(* CoDeSys 2.3.9.41 project: 5AxisMachine.pro *)
(* Libraries: TcUtilities.lib 10.1.13 20:12:12, TcBase.lib 14.5.09 12:14:08, TcSystem.lib 16.1.14 19:38:48, TcBaseMath.lib 27.7.04 12:07:56, TcMath.lib 23.9.04 15:15:30, TcMC2.lib 14.7.14 11:34:46, STANDARD.LIB 5.6.98 12:03:02, TcSUPS.lib 22.3.10 13:59:22, SysLibVisu.lib 7.7.04 18:17:22, SysLibTargetVisu.lib 16.6.08 16:24:26 *)

(* Task configuration *)
TASK Standard (PRIORITY := 0, INTERVAL := T#10ms);
	MAIN
END_TASK
TASK VISU_TASK (PRIORITY := 3, INTERVAL := T#200ms);
	MAINTARGETVISU_PAINT_CODE
END_TASK
TASK VISU_INPUT_TASK (PRIORITY := 2, INTERVAL := T#50ms);
	MAINTARGETVISU_INPUT_CODE
END_TASK

(* Global variable list: Global1_Persistent_Variables *)
VAR_GLOBAL PERSISTENT
	MachineRecipes				: ARRAY[1..NUMBER_OF_RECIPES] OF Recipe;
	nCurrentRecipe				: BYTE := 1; (* Current Machine Recipe *)
	nPartsCounter				: DWORD;


	VisuDoExecuteUserlevelInit 	: BOOL := TRUE;
	CurrentUserLevel 			: INT := 0;
	CurrentPasswords 			: ARRAY[0..7] OF STRING[20] := '','1','2','3','superuser4','8600','arl6','arl7'; (* Assigns Password Defaults *)
END_VAR

(* Global variable list: Global_Constant *)
VAR_GLOBAL CONSTANT
	NUMBER_OF_AXIS		: BYTE := 5;
	NUMBER_OF_MOVES 	: BYTE := 9;
	NUMBER_OF_RECIPES 	: BYTE := 25;
	CUTTER				: BYTE := 1;
	SIZER				: BYTE := 2;

	LEFT_HAND_SPINDLE	: BYTE := 1;
	RIGHT_HAND_SPINDLE	: BYTE := 2;
	CUTTER_AXIS			: BYTE := 3;
	CUTTER_SLIDE		: BYTE := 4;
	ENGAGE_AXIS			: BYTE := 5;

	SIZER_AXIS			: BYTE := 1;
	ARBOR_AXIS			: BYTE := 2;

	MAX_CYCLE_TIME		: WORD := 120;


	DEAFULT_AXIS_SPEED	: LREAL := 500;

	VERSION_NUMBER		: STRING :='V1.0.0 9_19_14';



END_VAR

(* Global variable list: Global_Variables *)
VAR_GLOBAL

(* IO Defined Here *)
	nRecipeNumber							   : BYTE; (* Holds Recipe Number for Editor *)

	Faults									   : Faults_STRUCT;
	Warnings								   : Warnings_STRUCT;

	nMachineType							   : BYTE := SIZER; (* Defines Machine Type 1 = Cutter, 2 = Sizer *)
	bAutomaticMode							   : BOOL;
END_VAR

(* Global variable list: Global_Variables_IO *)
VAR_GLOBAL
	(************ INPUTS ***********************)
	ibPowerOn						AT %I*		: BOOL;			(* True when power is on						*)
	ibLightScreenClear				AT %I*		: BOOL;			(* True when light screen is clear				*)
	ibCycleStartPB					AT %I*		: BOOL;			(* when true start machine cycle				*)
	ibLeftHandSpindleDriveOn		AT %I*		: BOOL;			(* When true left hand spindle is on			*)
	ibLeftHandSpindleDriveOK		AT %I*		: BOOL;			(* When true left hand spindle drive is faulted	*)
	ibRightHandSpindleDriveOn		AT %I*		: BOOL;			(* When true right hand spindle is on			*)
	ibRightHandSpindleDriveOK		AT %I*		: BOOL;			(* When true right hand spindle drive is faulted*)
	ibPartClampAdvanced				AT %I*		: BOOL;			(* When true the part clamp is clamped  		*)
	ibPartClampReturned				AT %I*		: BOOL;			(* When true the part clamp is returned 		*)
	ibPartClampLocked				AT %I*		: BOOL;			(* When true part clamp is in locked position	*)
	ibHydraulicsOverload			AT %I*		: BOOL;			(* Hydraulics overloaded when false				*)
	ibHydraulicsOverTemp			AT %I*		: BOOL;			(* Hydraulics over temp							*)
	ibHydraulicsLowLevel			AT %I*		: BOOL;			(* Hydraulics low level							*)

	(*************OUTPUTS***********************)

	qbLeftHandSpindleOn				AT %Q*		: BOOL;			(* Enable left hand spindle						*)
	qbRightHandSpindleOn			AT %Q*		: BOOL;			(* Enable right hand spindle					*)
	qbClosePartClampSolA			AT %Q*		: BOOL;			(* When true part clamp solenoid A closes clamp	*)
	qbOpenPartClampSolB				AT %Q*		: BOOL;			(* When trie part clamp solendoid B opens clamp *)
	qbSpareOutput					AT %Q*		: BOOL;
	qbOKToEnterGreenLamp			AT %Q*		: BOOL;
	qbMachineInCycleFaultRedLamp	AT %Q*		: BOOL;


END_VAR

(* Global variable list: TwinCAT_Configuration *)
(* Generated automatically by TwinCAT - (read only) *)
VAR_CONFIG
	MAIN.Axis_REF[1].PlcToNc AT %QB1 : PLCTONC_AXIS_REF;
	MAIN.Axis_REF[1].NcToPlc AT %IB6 : NCTOPLC_AXIS_REF;
	MAIN.Axis_REF[2].PlcToNc AT %QB129 : PLCTONC_AXIS_REF;
	MAIN.Axis_REF[2].NcToPlc AT %IB134 : NCTOPLC_AXIS_REF;
	MAIN.Axis_REF[3].PlcToNc AT %QB257 : PLCTONC_AXIS_REF;
	MAIN.Axis_REF[3].NcToPlc AT %IB262 : NCTOPLC_AXIS_REF;
	MAIN.Axis_REF[4].PlcToNc AT %QB385 : PLCTONC_AXIS_REF;
	MAIN.Axis_REF[4].NcToPlc AT %IB390 : NCTOPLC_AXIS_REF;
	MAIN.Axis_REF[5].PlcToNc AT %QB513 : PLCTONC_AXIS_REF;
	MAIN.Axis_REF[5].NcToPlc AT %IB518 : NCTOPLC_AXIS_REF;
	.ibPowerOn AT %IX648.0 : BOOL;	(*  ~ {LinkedWith:TIID^Device 1 (EtherCAT)^Term 1 (EK1200)^Term 2 (EL1809)^Channel 1^Power On} *)
	.ibLightScreenClear AT %IX648.1 : BOOL;	(*  ~ {LinkedWith:TIID^Device 1 (EtherCAT)^Term 1 (EK1200)^Term 2 (EL1809)^Channel 2^Light Curtain Clear} *)
	.ibCycleStartPB AT %IX648.2 : BOOL;	(*  ~ {LinkedWith:TIID^Device 1 (EtherCAT)^Term 1 (EK1200)^Term 2 (EL1809)^Channel 3^Cycle Start} *)
	.ibLeftHandSpindleDriveOn AT %IX648.3 : BOOL;
	.ibLeftHandSpindleDriveOK AT %IX648.4 : BOOL;
	.ibRightHandSpindleDriveOn AT %IX648.5 : BOOL;
	.ibRightHandSpindleDriveOK AT %IX648.6 : BOOL;
	.ibPartClampAdvanced AT %IX648.7 : BOOL;	(*  ~ {LinkedWith:TIID^Device 1 (EtherCAT)^Term 1 (EK1200)^Term 2 (EL1809)^Channel 4^Part Clamp Closed} *)
	.ibPartClampReturned AT %IX649.0 : BOOL;	(*  ~ {LinkedWith:TIID^Device 1 (EtherCAT)^Term 1 (EK1200)^Term 2 (EL1809)^Channel 5^Part Clamp Open} *)
	.ibPartClampLocked AT %IX649.1 : BOOL;
	.ibHydraulicsOverload AT %IX649.2 : BOOL;
	.ibHydraulicsOverTemp AT %IX652.0 : BOOL;
	.ibHydraulicsLowLevel AT %IX652.1 : BOOL;
	.qbLeftHandSpindleOn AT %QX644.0 : BOOL;
	.qbRightHandSpindleOn AT %QX644.1 : BOOL;
	.qbClosePartClampSolA AT %QX644.2 : BOOL;
	.qbOpenPartClampSolB AT %QX644.3 : BOOL;
	.qbSpareOutput AT %QX644.4 : BOOL;
	.qbOKToEnterGreenLamp AT %QX644.5 : BOOL;	(*  ~ {LinkedWith:TIID^Device 1 (EtherCAT)^Term 1 (EK1200)^Term 3 (EL2828)^Channel 7^Green Lamp (OK To Enter)} *)
	.qbMachineInCycleFaultRedLamp AT %QX644.6 : BOOL;	(*  ~ {LinkedWith:TIID^Device 1 (EtherCAT)^Term 1 (EK1200)^Term 3 (EL2828)^Channel 8^Red Lamp (Faulted)} *)
END_VAR

(* Data type *)
TYPE AXISSEQUENCE :
(
	AXIS_INIT,
	AXIS_RESET,
	AXIS_FAULTED,
	AXIS_READY,
	AXIS_POWER_ON,
	AXIS_STOP,
	AXIS_HOMING,
	AXIS_HOMED,
	AXIS_RUNNING
);

END_TYPE

(* Data type *)
TYPE FAULTS_STRUCT :
STRUCT
	bOperator_Stop					: BOOL; (* True when operate stops the machine							*)
	bLeftHandSpindleVFDError		: BOOL; (* True when left hand spindle VFD is at Fault					*)
	bRightHandSpindleVFDError		: BOOL;
	bProgramError					: BOOL;
	bLeftSpindleServoError			: BOOL;
	bRightSpindlervoError			: BOOL;
	bCutterServorError				: BOOL;
	bCutterSlideServoError			: BOOL;
	bEngageServoError				: BOOL;
	bCycleTimeExceeded				: BOOL; (* True when the cycle time took too long to complete			*)
END_STRUCT
END_TYPE

(* Data type *)
TYPE MACHINE_SEQUENCE :
(
	MACHINE_INIT,
	MACHINE_RESET,
	MACHINE_FAULTED,
	MACHINE_READY,
	ENABLE_SERVOS,
	MOVE_TO_END_CUT,
	MOVE_TO_START_SIZER,
	POSITION_SIZER_SERVOS,
	MOVE_TO_CRUSHED_POSITION,
	MOVE_SIZER_TO_RELIEVED_POSITION,
	MOVE_SIZER_TO_UNLOAD,
	RETURN_SIZER,
	MOVE_TO_FIRST_CUT,
	COUPLE_DRIVES,
	DECOUPLE_DRIVES,
	OPERATE_FIRST_CUT,
	MOVE_TO_NEXT_CUT,
	ADVANCE_ENGAGE,
	RETURN_ENGAGE,
	OPERATE_CUT,
	RETRACT_FROM_CUT,
	RETURN_MACHINE
);

END_TYPE

(* Data type *)
TYPE RECIPE :
STRUCT

	bPartClampEnable		: BOOL;											(* When true part clamp is enabled						*)
	arrAxis1MoveTable		: ARRAY[1..NUMBER_OF_MOVES] OF LREAL;			(* Left Spindle Axis move table							*)
	arrAxis2MoveTable		: ARRAY[1..NUMBER_OF_MOVES] OF LREAL;			(* Right spindle move table								*)
	arrAxis3MoveTable		: ARRAY[1..2] OF LREAL;							(* Cutter move table									*)
	arrAxis4MoveTable		: ARRAY[1..NUMBER_OF_MOVES] OF LREAL;			(* Cutter slide move table								*)
	arrAxis5MoveTable		: ARRAY[1..2] OF LREAL;							(* Engage move table									*)
	Axis1HomePosition		: LREAL;										(* Axis 1 Home Position									*)
	nNumberOfCuts			: BYTE;											(* Number of cuts to be made							*)
	timeCutterTimer			: TIME;											(* Cutter Timer Time									*)
	rAxis1Speed				: LREAL;										(* Speed of Axis #1										*)
	rAxis2Speed				: LREAL;										(* Speed of Axis #2										*)
	rAxis3Speed				: LREAL;										(* Speed of Axis #3										*)
	rAxis4Speed				: LREAL;										(* Speed of Axis #4										*)
	rAxis5Speed				: LREAL;										(* Speed of Axis #5										*)
	nNumberOfCycles			: BYTE; 										(* Number of cycles of the sizer						*)
	sRecipeName				: STRING;										(* Part Type Description								*)
END_STRUCT
END_TYPE

(* Data type *)
TYPE WARNINGS_STRUCT :
STRUCT
	bHopperLow						: BOOL;
	bConveyorFull					: BOOL;
END_STRUCT
END_TYPE

(* POU MAIN, LD *)
(********************************************************************************************************
NAME...........	:	Main Program
DATE...........	:	08.6.2014
AUTHOR.........	:	ARL

DESCRIPTION....	:	Handling of main routine for the Machine.

HISTORY:	
08.6.2014	v1.0.0	GPK	Start coding
*********************************************************************************************************)
PROGRAM MAIN
VAR_INPUT
	nTargetPosition 			: ARRAY[1..NUMBER_OF_AXIS] OF LREAL;
	nMoveVelocity   			: ARRAY[1..NUMBER_OF_AXIS] OF LREAL;
	bClosePartClamp				: BOOL;
	bMoveAbsolute				: ARRAY[1..NUMBER_OF_AXIS] OF BOOL;
	bAxisEnable 				: ARRAY[1..NUMBER_OF_AXIS] OF BOOL;


	bLeftHandSpindleRun			: BOOL;
	bRightHandSpindleRun		: BOOL;

	bCoupleAxis					: BOOL;
	bDeCoupleAxis				: BOOL;
	bAxis2Coupled				: BOOL;
	bAxis4Coupled				: BOOL;
	bInCycle					: BOOL;

	bJogAxisForward				: ARRAY[1..NUMBER_OF_AXIS] OF BOOL;
	bJogAxisReverse				: ARRAY[1..NUMBER_OF_AXIS] OF BOOL;
	bFaultPresent				: BOOL;
END_VAR
VAR
	Axis						: ARRAY[1..NUMBER_OF_AXIS] OF FB_Motion;

	Axis_REF					: ARRAY[1..NUMBER_OF_AXIS] OF AXIS_REF;

	bAxisHasError				: ARRAY[1..NUMBER_OF_AXIS] OF BOOL;
	bMoveRelative				: ARRAY[1..NUMBER_OF_AXIS] OF BOOL;
	bMoveComplete				: ARRAY[1..NUMBER_OF_AXIS] OF BOOL;
	bPowerOnActive				: ARRAY[1..NUMBER_OF_AXIS] OF BOOL;


	sSequenceText				: ARRAY[1..NUMBER_OF_AXIS] OF STRING;
	loop						: BYTE; (* Used to loop through all axis *)
	bResetLoop					: BOOL;


	bStartMachine				: BOOL;
	bStopMachine				: BOOL;
	bReset						: BOOL;
	bMachineRunning				: BOOL;





	ToggleLamp					: FB_Toggle; 			(* FB to toggle variable or output off/on   *)
	LeftHandSpindleMotor		: FB_Motor_Ctrl; 		(* FB for simple motor control 				*)
	RightHandSpindleMotor		: FB_Motor_Ctrl; 		(* FB for simple motor control 				*)
	PartClamp					: FB_CylinderControl;	(* FB To Operate Part Clamp					*)

	ctCycleCounter				: CTU;
	wCounterPreset				: WORD; (* Some Comment *)


	bResetCounter				: BOOL;		(*Reset Counter*)
	bTriggerCounter				: BOOL;
	CounterDone					: BOOL;
	bStartButtonIndicator		: BOOL;
	bResetTimeCounter			: BOOL;


	CoupleAxis2					: FB_CoupleAxis;
	CoupleAxis4					: FB_CoupleAxis;

	tmrCycleTimer				: TON;

	cntSecondsCounter			: CTU;
	re_InCycle					: R_TRIG;
	nCycleTime					: WORD;

END_VAR
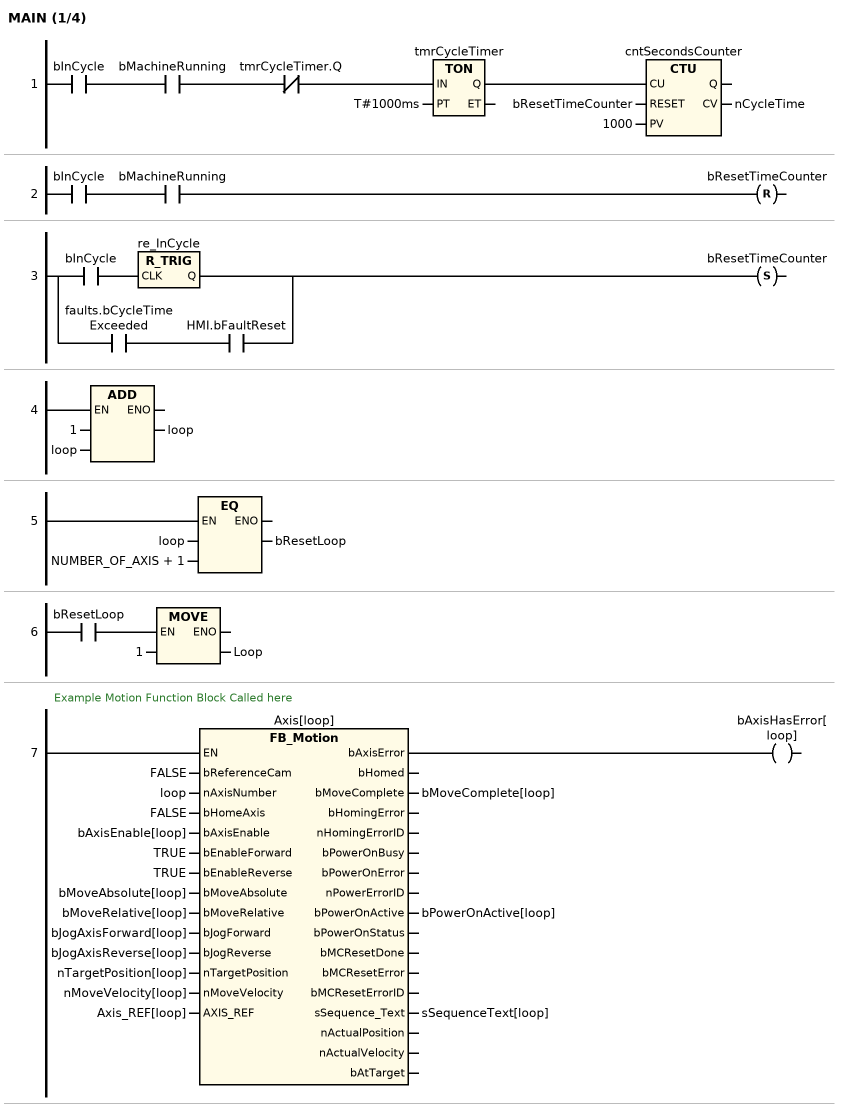
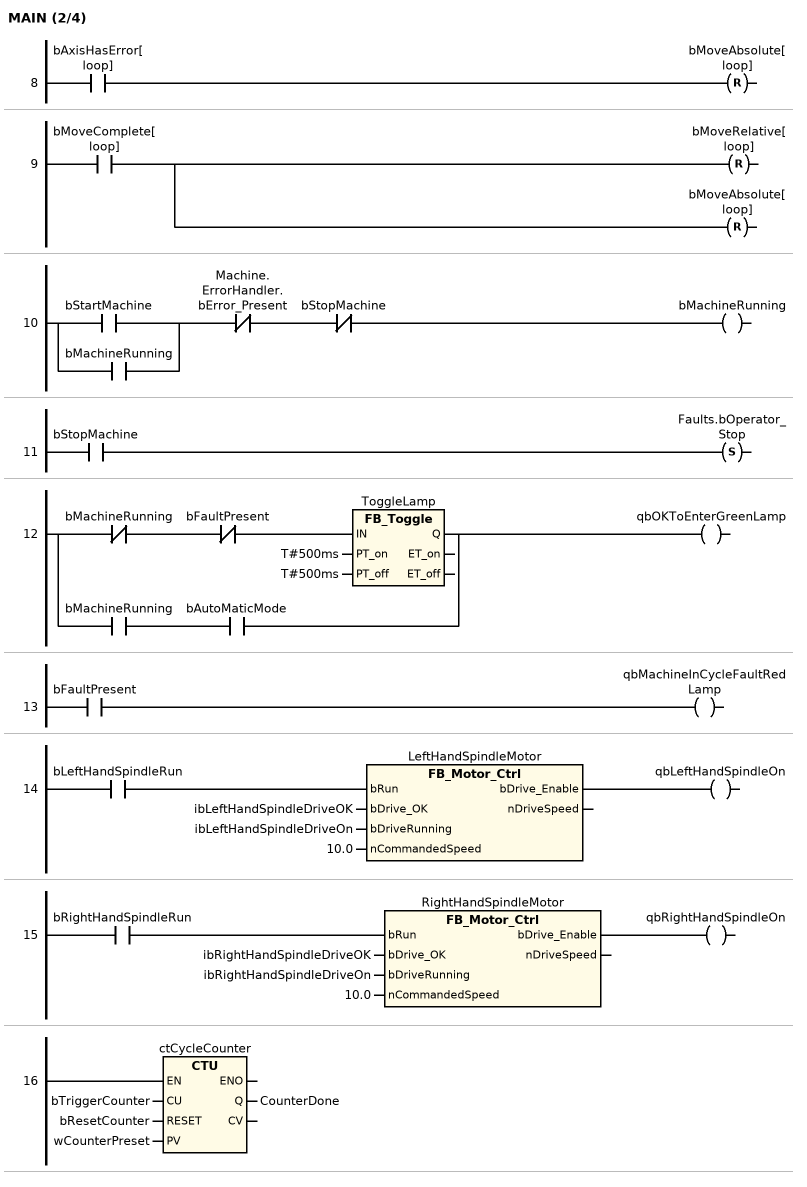
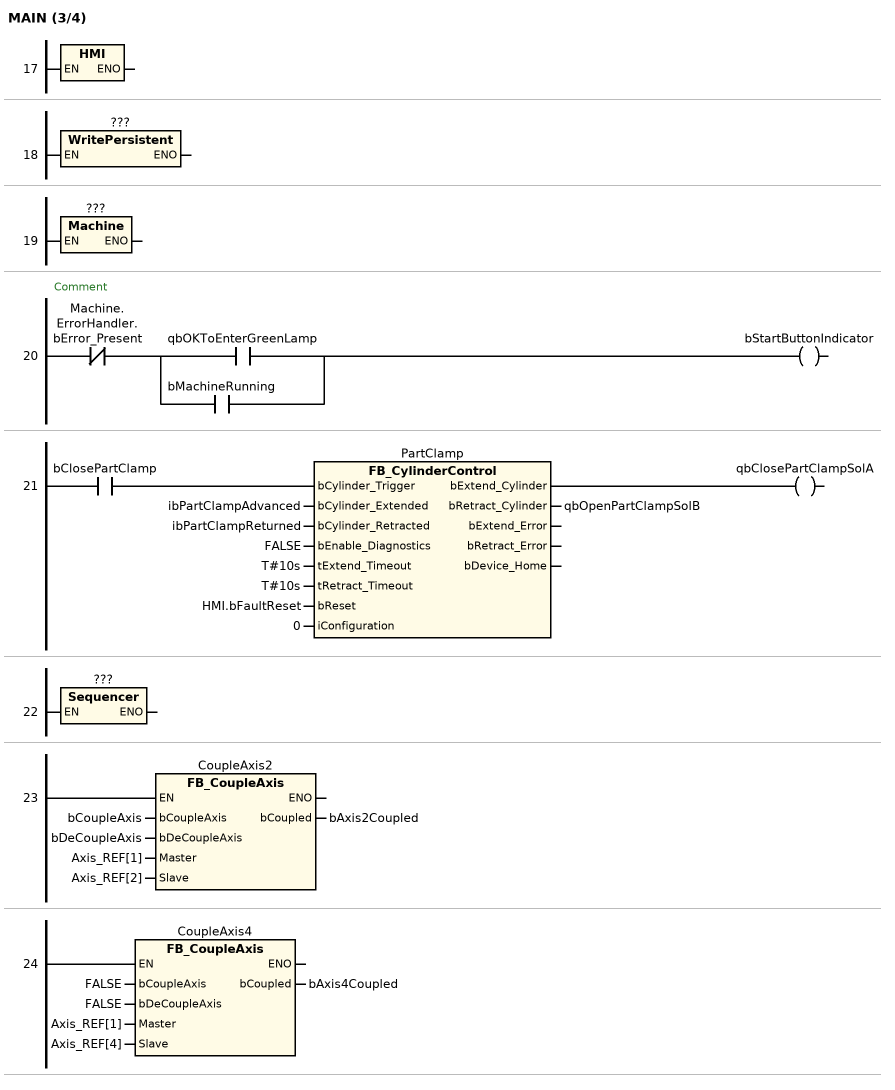
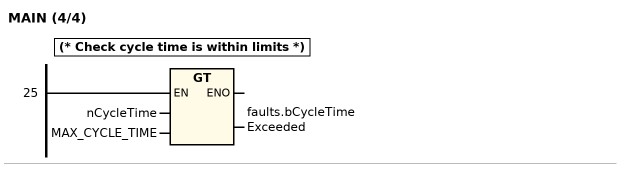
_LD_ (* Ladder Diagram *)
NETWORK 1
	[bInCycle] - [bMachineRunning] - [/tmrCycleTimer.Q] - tmrCycleTimer:TON(IN: *, PT: T#1000ms) - cntSecondsCounter:CTU(CU: *, RESET: bResetTimeCounter, PV: 1000, CV => nCycleTime)
NETWORK 2
	[bInCycle] - [bMachineRunning] --- (R bResetTimeCounter)
NETWORK 3
	{ [bInCycle] - re_InCycle:R_TRIG(CLK: *) | [faults.bCycleTimeExceeded] - [HMI.bFaultReset] } --- (S bResetTimeCounter)
NETWORK 4
	*
		EN --- ADD(1, loop) => loop
NETWORK 5
	*
		EN --- EQ(loop, NUMBER_OF_AXIS + 1) => bResetLoop
NETWORK 6
	[bResetLoop]
		EN --- MOVE(1) => Loop
NETWORK 7 (* Example Motion Function Block Called here *)
	Axis[loop]:FB_Motion(EN: *, bReferenceCam: FALSE, nAxisNumber: loop, bHomeAxis: FALSE, bAxisEnable: bAxisEnable[loop], bEnableForward: TRUE, bEnableReverse: TRUE, bMoveAbsolute: bMoveAbsolute[loop], bMoveRelative: bMoveRelative[loop], bJogForward: bJogAxisForward[loop], bJogReverse: bJogAxisReverse[loop], nTargetPosition: nTargetPosition[loop], nMoveVelocity: nMoveVelocity[loop], AXIS_REF: Axis_REF[loop], bMoveComplete => bMoveComplete[loop], bPowerOnActive => bPowerOnActive[loop], sSequence_Text => sSequenceText[loop]) --- (bAxisHasError[loop])
NETWORK 8
	[bAxisHasError[loop]] --- (R bMoveAbsolute[loop])
NETWORK 9
	[bMoveComplete[loop]] --- (R bMoveRelative[loop]) (R bMoveAbsolute[loop])
NETWORK 10
	{ [bStartMachine] | [bMachineRunning] } - [/Machine.ErrorHandler.bError_Present] - [/bStopMachine] --- (bMachineRunning)
NETWORK 11
	[bStopMachine] --- (S Faults.bOperator_Stop)
NETWORK 12
	{ [/bMachineRunning] - [/bFaultPresent] - ToggleLamp:FB_Toggle(IN: *, PT_on: T#500ms, PT_off: T#500ms) | [bMachineRunning] - [bAutoMaticMode] } --- (qbOKToEnterGreenLamp)
NETWORK 13
	[bFaultPresent] --- (qbMachineInCycleFaultRedLamp)
NETWORK 14
	[bLeftHandSpindleRun] - LeftHandSpindleMotor:FB_Motor_Ctrl(bRun: *, bDrive_OK: ibLeftHandSpindleDriveOK, bDriveRunning: ibLeftHandSpindleDriveOn, nCommandedSpeed: 10.0) --- (qbLeftHandSpindleOn)
NETWORK 15
	[bRightHandSpindleRun] - RightHandSpindleMotor:FB_Motor_Ctrl(bRun: *, bDrive_OK: ibRightHandSpindleDriveOK, bDriveRunning: ibRightHandSpindleDriveOn, nCommandedSpeed: 10.0) --- (qbRightHandSpindleOn)
NETWORK 16
	*
		EN --- ctCycleCounter:CTU(CU: bTriggerCounter, RESET: bResetCounter, PV: wCounterPreset) => CounterDone
NETWORK 17
	*
		EN --- HMI()
NETWORK 18
	*
		EN --- ???:WritePersistent()
NETWORK 19
	*
		EN --- ???:Machine()
NETWORK 20 (* Comment *)
	[/Machine.ErrorHandler.bError_Present] - { [qbOKToEnterGreenLamp] | [bMachineRunning] } --- (bStartButtonIndicator)
NETWORK 21
	[bClosePartClamp] - PartClamp:FB_CylinderControl(bCylinder_Trigger: *, bCylinder_Extended: ibPartClampAdvanced, bCylinder_Retracted: ibPartClampReturned, bEnable_Diagnostics: FALSE, tExtend_Timeout: T#10s, tRetract_Timeout: T#10s, bReset: HMI.bFaultReset, iConfiguration: 0, bRetract_Cylinder => qbOpenPartClampSolB) --- (qbClosePartClampSolA)
NETWORK 22
	*
		EN --- ???:Sequencer()
NETWORK 23
	*
		EN --- CoupleAxis2:FB_CoupleAxis(bCoupleAxis: bCoupleAxis, bDeCoupleAxis: bDeCoupleAxis, Master: Axis_REF[1], Slave: Axis_REF[2]) => bAxis2Coupled
NETWORK 24
	*
		EN --- CoupleAxis4:FB_CoupleAxis(bCoupleAxis: FALSE, bDeCoupleAxis: FALSE, Master: Axis_REF[1], Slave: Axis_REF[4]) => bAxis4Coupled
NETWORK 25 (* Check cycle time is within limits *):
	*
		EN --- GT(nCycleTime, MAX_CYCLE_TIME) => faults.bCycleTimeExceeded
_END_LD_
(* the same logic as Structured Text *)
(* Network 1 *)
tmrCycleTimer(IN := bInCycle AND bMachineRunning AND NOT tmrCycleTimer.Q, PT := T#1000ms);
cntSecondsCounter(CU := tmrCycleTimer.Q, RESET := bResetTimeCounter, PV := 1000);
nCycleTime := cntSecondsCounter.CV;
(* Network 2 *)
IF bInCycle AND bMachineRunning THEN bResetTimeCounter := FALSE; END_IF;
(* Network 3 *)
re_InCycle(CLK := bInCycle);
IF re_InCycle.Q OR faults.bCycleTimeExceeded AND HMI.bFaultReset THEN bResetTimeCounter := TRUE; END_IF;
(* Network 4 *)
loop := 1 + loop;
(* Network 5 *)
bResetLoop := loop = (NUMBER_OF_AXIS + 1);
(* Network 6 *)
IF bResetLoop THEN
	Loop := 1;
END_IF;
(* Network 7 *)
Axis[loop](EN := TRUE, bReferenceCam := FALSE, nAxisNumber := loop, bHomeAxis := FALSE, bAxisEnable := bAxisEnable[loop], bEnableForward := TRUE, bEnableReverse := TRUE, bMoveAbsolute := bMoveAbsolute[loop], bMoveRelative := bMoveRelative[loop], bJogForward := bJogAxisForward[loop], bJogReverse := bJogAxisReverse[loop], nTargetPosition := nTargetPosition[loop], nMoveVelocity := nMoveVelocity[loop], AXIS_REF := Axis_REF[loop]);
bMoveComplete[loop] := Axis[loop].bMoveComplete;
bPowerOnActive[loop] := Axis[loop].bPowerOnActive;
sSequenceText[loop] := Axis[loop].sSequence_Text;
bAxisHasError[loop] := Axis[loop].bAxisError;
(* Network 8 *)
IF bAxisHasError[loop] THEN bMoveAbsolute[loop] := FALSE; END_IF;
(* Network 9 *)
IF bMoveComplete[loop] THEN bMoveRelative[loop] := FALSE; bMoveAbsolute[loop] := FALSE; END_IF;
(* Network 10 *)
bMachineRunning := (bStartMachine OR bMachineRunning) AND NOT Machine.ErrorHandler.bError_Present AND NOT bStopMachine;
(* Network 11 *)
IF bStopMachine THEN Faults.bOperator_Stop := TRUE; END_IF;
(* Network 12 *)
ToggleLamp(IN := NOT bMachineRunning AND NOT bFaultPresent, PT_on := T#500ms, PT_off := T#500ms);
qbOKToEnterGreenLamp := ToggleLamp.Q OR bMachineRunning AND bAutoMaticMode;
(* Network 13 *)
qbMachineInCycleFaultRedLamp := bFaultPresent;
(* Network 14 *)
LeftHandSpindleMotor(bRun := bLeftHandSpindleRun, bDrive_OK := ibLeftHandSpindleDriveOK, bDriveRunning := ibLeftHandSpindleDriveOn, nCommandedSpeed := 10.0);
qbLeftHandSpindleOn := LeftHandSpindleMotor.bDrive_Enable;
(* Network 15 *)
RightHandSpindleMotor(bRun := bRightHandSpindleRun, bDrive_OK := ibRightHandSpindleDriveOK, bDriveRunning := ibRightHandSpindleDriveOn, nCommandedSpeed := 10.0);
qbRightHandSpindleOn := RightHandSpindleMotor.bDrive_Enable;
(* Network 16 *)
ctCycleCounter(CU := bTriggerCounter, RESET := bResetCounter, PV := wCounterPreset);
CounterDone := ctCycleCounter.Q;
(* Network 17 *)
HMI();
(* Network 18: see the listing above *)
(* Network 19: see the listing above *)
(* Network 20 *)
bStartButtonIndicator := NOT Machine.ErrorHandler.bError_Present AND (qbOKToEnterGreenLamp OR bMachineRunning);
(* Network 21 *)
PartClamp(bCylinder_Trigger := bClosePartClamp, bCylinder_Extended := ibPartClampAdvanced, bCylinder_Retracted := ibPartClampReturned, bEnable_Diagnostics := FALSE, tExtend_Timeout := T#10s, tRetract_Timeout := T#10s, bReset := HMI.bFaultReset, iConfiguration := 0);
qbOpenPartClampSolB := PartClamp.bRetract_Cylinder;
qbClosePartClampSolA := PartClamp.bExtend_Cylinder;
(* Network 22: see the listing above *)
(* Network 23 *)
CoupleAxis2(bCoupleAxis := bCoupleAxis, bDeCoupleAxis := bDeCoupleAxis, Master := Axis_REF[1], Slave := Axis_REF[2]);
bAxis2Coupled := CoupleAxis2.bCoupled;
(* Network 24 *)
CoupleAxis4(bCoupleAxis := FALSE, bDeCoupleAxis := FALSE, Master := Axis_REF[1], Slave := Axis_REF[4]);
bAxis4Coupled := CoupleAxis4.bCoupled;
(* Network 25 *)
faults.bCycleTimeExceeded := nCycleTime > MAX_CYCLE_TIME;
END_PROGRAM

(* POU Motion/FB_Motion, ST *)
(********************************************************************************************************

NAME...........	:	FB_Motion
DATE...........	:	7/23/2014
AUTHOR.........	:	Graeme Peek Beckhoff Automation

DESCRIPTION....	:	Motion Axis Control Function Block
					NOTE: Given as is as an example, if used as part of a working machine then it must be validated and adjusted as required.
					Beckhoff assumes no responsability for the accuracy of this software.

HISTORY:	
5/23/2014	v1.0.0	Graeme	Start coding
*************************************************************************************************************)
FUNCTION_BLOCK FB_Motion
VAR_INPUT
	EN						: BOOL;						(* Block enabled when true							*)
	bReferenceCam			: BOOL; 					(* True when reference cam is on 					*)
	nAxisNumber				: BYTE;						(* Holds Axis Number								*)
	bHomeAxis				: BOOL;						(* When true homing is initiated					*)
	bAxisEnable				: BOOL;						(* When true then enable this axis					*)
	bEnableForward			: BOOL;
	bEnableReverse			: BOOL;
	bMoveAbsolute			: BOOL;
	bMoveRelative			: BOOL;
	bJogForward				: BOOL;						(* When true axis jogs forward						*)
	bJogReverse				: BOOL;						(* When true axis jogs in reverse					*)
	nTargetPosition			: LREAL;
	nMoveVelocity			: LREAL;
END_VAR
VAR_OUTPUT
	bAxisError				: BOOL;
	bHomed					: BOOL;						(* True when axis has homed							*)
	bMoveComplete			: BOOL;						(* True when any move has completed					*)
	bHomingError			: BOOL;						(* True when an error ocurred to the homing FB		*)
	nHomingErrorID			: UDINT;					(* Holds homing FB error code						*)
	bPowerOnBusy			: BOOL;						(* True when power is on 							*)
	bPowerOnError			: BOOL;						(* True if an error occurred turing axis power on	*)
	nPowerErrorID			: UDINT;					(* Holds error code for power on command			*)
	bPowerOnActive			: BOOL;						(* True when power is FB is called					*)
	bPowerOnStatus			: BOOL;						(* True when axis is ready 							*)
	bMCResetDone			: BOOL;						(* True when MC Reset command has completed			*)
	bMCResetError			: BOOL;						(* True when error occurred during MC Reset			*)
	bMCResetErrorID			: UDINT;					(* Holds error code for MC Reset Command			*)
	sSequence_Text			: STRING;
	nActualPosition			: LREAL;					(* Holds actual axis position						*)
	nActualVelocity			: LREAL; 					(* Holds actual Velocity of axis					*)
	bAtTarget				: BOOL;						(* True when current position is at the target pos. *)
END_VAR
VAR
	(* Declare All Motion Function Blocks 	*)
	MC_PowerOn				: MC_Power;					(* Power On FB 										*)
	MC_Reset				: MC_Reset;					(* Reset Axis FB									*)
	MC_Home					: MC_Home;					(* Homing Axis FB									*)
	MC_AbsoluteMove			: MC_MoveAbsolute;			(* Move Absolute Handler							*)
	MC_RelativeMove			: MC_MoveRelative;			(* Move Relative Handler							*)
	MC_Jog					: MC_Jog;					(* Jog Axis Handler									*)

	(* Declare Local Variables				*)
	bHomeExecute			: BOOL;						(* When true homing is executed						*)
	bPowerExecute			: BOOL;						(* When true power on is executed					*)
	bAxisResetExecute		: BOOL;
	bAxisMoveRelativeExecute: BOOL;
	bAxisAbsoluteExecute	: BOOL;
	bNoFaults				: BOOL;
	bResetFault				: BOOL;
	bHomingDone				: BOOL;

	bAxisPowerBusy			: BOOL;
	bAxisPowerError			: BOOL;
	nFaultCode				: UDINT;
	nSequence				: AxisSequence;				(* Holds motion FB sequence State					*)

END_VAR

VAR_IN_OUT
	AXIS_REF				: AXIS_REF;
END_VAR
(* Call All MC2 Drive Motion Function Blocks *)
MC_Home(
	Execute:= bHomeExecute,
	Position:= ,
	HomingMode:= ,
	bCalibrationCam:= bReferenceCam ,
	Axis:= AXIS_REF,
	Done=> bHomingDone,
	Error=> bHomingError,
	ErrorID=> nHomingErrorID);


IF nHomingErrorID > 0 THEN
	nFaultCode := nHomingErrorID;
ELSIF nPowerErrorID > 0 THEN
	nFaultCode := nPowerErrorID;
ELSIF bMCResetErrorID > 0 THEN
	nFaultCode := bMCResetErrorID;
ELSIF MC_AbsoluteMove.ErrorID > 0 THEN
	nFaultCode := MC_AbsoluteMove.ErrorID;
END_IF;

(* Reset Error Code if no errors found *)
IF nHomingErrorID = 0 AND nPowerErrorID = 0 AND bMCResetErrorID = 0
	AND MC_AbsoluteMove.ErrorID = 0 THEN
	nFaultCode := 0;
END_IF;


MC_PowerOn(
	Enable:= bPowerExecute,
	Enable_Positive:= bEnableForward,
	Enable_Negative:= bEnableReverse,
	Axis:= AXIS_REF ,
	Status=> bPowerOnStatus,
	Busy=> bPowerOnBusy,
	Active=>bPowerOnActive ,
	Error=> bPowerOnError ,
	ErrorID=> nPowerErrorID );

MC_Reset(
	Execute:= bAxisResetExecute,
	Axis:= AXIS_REF,
	Done=> ,
	Busy=>bMCResetDone ,
	Error=>bMCResetError ,
	ErrorID=>bMCResetErrorID );

MC_RelativeMove(
	Execute:= bMoveRelative ,
	Distance:= nTargetPosition ,
	Velocity:= nTargetPosition,
	Axis:= AXIS_REF,
	Done=> ,
	Busy=> ,
	Active=> ,
	CommandAborted=> ,
	Error=> ,
	ErrorID=> );

MC_AbsoluteMove(
	Execute:= bMoveAbsolute,
	Position:= nTargetPosition ,
	Velocity:= nMoveVelocity ,
	Axis:= AXIS_REF ,
	Done=> ,
	Busy=> ,
	Active=> ,
	CommandAborted=> ,
	Error=> ,
	ErrorID=> );

MC_Jog(
	JogForward:= bJogForward,
	JogBackwards:= bJogReverse ,
	Mode:= ,
	Position:= ,
	Velocity:= nMoveVelocity,
	Axis:= AXIS_REF,
	Done=> ,
	Busy=> ,
	Active=> ,
	CommandAborted=> ,
	Error=> ,
	ErrorID=> );

sSequence_Text := GetMotionSequenceActionDescription(iSequence_state := nSequence);

nActualPosition := AXIS_REF.NcToPlc.ActPos;
nActualVelocity	:= AXIS_REF.NcToPlc.ActVelo;

IF MC_AbsoluteMove.Done OR MC_RelativeMove.Done THEN
	bMoveComplete := TRUE;
ELSE
	bMoveComplete := FALSE;
END_IF;

IF (nActualPosition > (nTargetPosition - 5)) AND (nActualPosition < (nTargetPosition + 5)) THEN
	bAtTarget := TRUE;
ELSE
	bAtTarget := FALSE;
END_IF;

CASE nSequence OF
		AXIS_INIT :
			bAxisResetExecute 				:= FALSE;
			bAxisMoveRelativeExecute 		:= FALSE;
			bAxisAbsoluteExecute 			:= FALSE;
			bHomeExecute			 		:= FALSE;
			bPowerExecute					:= FALSE;
			bAxisError						:= FALSE;
			IF (NOT bHomeAxis) THEN
				bHomed						:= FALSE;
			END_IF;
			IF EN THEN
				nSequence 					:= AXIS_RESET;
			END_IF;

		AXIS_RESET:
			bAxisResetExecute 		 		:= TRUE;
			IF MC_Reset.Done THEN
				bAxisResetExecute 			:= FALSE;
				nSequence					:= AXIS_READY;
			END_IF

		AXIS_FAULTED:
			bNoFaults 		:= FALSE;
			bAxisError		:= TRUE;

			IF bResetFault AND (NOT bAxisEnable) THEN
				nSequence 	:= AXIS_INIT;
			END_IF

		AXIS_READY:
			(* Once axis is enabled move to power on axis *)
			IF bAxisEnable THEN
				nSequence 		:= AXIS_POWER_ON;
			END_IF

		AXIS_POWER_ON:
			bPowerExecute	:= TRUE;
			(* Once Power on has completed move on to homing or running *)
			IF bPowerOnStatus AND (NOT bAxisPowerError) THEN
				IF bHomeAxis AND (NOT bHomed) THEN
					nSequence := AXIS_HOMING;
				ELSE
					nSequence := AXIS_RUNNING;
				END_IF;
			END_IF
			(* If error during power up then flag a fault *)
			IF bAxisPowerError THEN
				nSequence := AXIS_FAULTED;
				bPowerExecute := FALSE;
			END_IF

		AXIS_STOP:
			;

		AXIS_HOMING:
			bHomed 			:= FALSE; (* Reset axis homed flag *)
			bHomeExecute 	:= TRUE; (* Turn on homing *)
			(* Once homed move to axis is homed state *)
			IF bHomingDone THEN
				nSequence := AXIS_HOMED;
			END_IF
			(* If an error occurss during homing then flag a fault *)
			IF MC_Home.Error THEN
				nSequence := AXIS_FAULTED;
				bHomeExecute := FALSE;
			END_IF

		AXIS_HOMED:
			bHomeExecute := FALSE; (* Turn off homing *)
			bHomed := TRUE;
		    nSequence := AXIS_RUNNING;

		AXIS_RUNNING:
			IF MC_RelativeMove.Done THEN
				bAxisMoveRelativeExecute := FALSE;
			END_IF
			IF MC_AbsoluteMove.Done THEN
				bAxisAbsoluteExecute := FALSE;
			END_IF

			IF MC_AbsoluteMove.Error THEN
				nSequence := AXIS_FAULTED;
			END_IF;
	END_CASE

(* IF Axis is NOT enabled THEN reset the sequence*)
IF (NOT bAxisEnable) AND (nSequence > AXIS_READY)  THEN
	nSequence := AXIS_INIT;
END_IF

IF nFaultCode > 0 AND NOT bResetFault THEN
	bNoFaults  := FALSE;
	nSequence := AXIS_FAULTED;
END_IF;
END_FUNCTION_BLOCK

(* POU Motion/GetMotionSequenceActionDescription, ST *)
(********************************************************************************************************
NAME...........	:	GetMotionSequenceActionDescription
DATE...........	:	06.04.2014
AUTHOR.........	:	Graeme Peek (Beckhoff Automation)

DESCRIPTION....	:	Function to assign meaningful text to action text based on current action

HISTORY:	
06.04.2014	v1.0.0	GPK	Start coding
*********************************************************************************************************)
FUNCTION GetMotionSequenceActionDescription : STRING
VAR_INPUT
	iSequence_State 			: AxisSequence;
END_VAR
VAR
END_VAR
CASE iSequence_State OF

	AXIS_INIT: 		GetMotionSequenceActionDescription := 'Initialising Axis';
	AXIS_RESET:		GetMotionSequenceActionDescription := 'Resettng Axis';
	AXIS_READY:		GetMotionSequenceActionDescription := 'Axis Ready';
	AXIS_POWER_ON:	GetMotionSequenceActionDescription := 'Powering On Axis';
	AXIS_FAULTED:	GetMotionSequenceActionDescription := 'Axis Faulted';
	AXIS_STOP:		GetMotionSequenceActionDescription := 'Axis Stopped';
	AXIS_HOMING:	GetMotionSequenceActionDescription := 'Axis Homing';
	AXIS_HOMED:		GetMotionSequenceActionDescription := 'Axis Homed';
	AXIS_RUNNING:	GetMotionSequenceActionDescription := 'Axis Running';
ELSE
	GetMotionSequenceActionDescription := 'Unknown Sequence State';
END_CASE
END_FUNCTION

(* POU Standard FB's/FB_Toggle, ST *)
(********************************************************************************************************
NAME...........	:	Toggle Function Block.
DATE...........	:	08.6.2010
AUTHOR.........	:	Graeme Peek 

DESCRIPTION....	:	Toggles output when enabled based on time given.
					Inputs:
						enable : Bool; When High function runs toggling output
						rate   : Time; Number of ms or seconds between state changes.
					Outputs:
						toggle_output : bool; The output value of function.
HISTORY:	
08.11.2014	v1.1.0	GPK	Start coding
*********************************************************************************************************)
FUNCTION_BLOCK FB_Toggle
VAR_INPUT
	IN				: BOOL;
	PT_on			: TIME;
	PT_off			: TIME;
END_VAR
VAR_OUTPUT
	Q				: BOOL;
	ET_on			: TIME;
	ET_off			: TIME;
END_VAR
VAR
	toggle_timer_on				: TON;
	toggle_timer_off			: TOF;
END_VAR
(* Call Timers *)
toggle_timer_off(PT:=PT_off, ET => ET_off );
toggle_timer_on(PT:= PT_on, ET => ET_on );

(* If enable is high start timers *)
IF IN THEN
	IF (NOT toggle_timer_off.Q) THEN
		toggle_timer_off.IN := TRUE;
		toggle_timer_on.IN  := TRUE;
		Q := FALSE;
	ELSIF toggle_timer_on.Q THEN
		toggle_timer_off.IN := FALSE;
		toggle_timer_on.IN  := FALSE;
		Q := TRUE;
	END_IF;
ELSE
	(* Ensure all timers are off and output is off *)
	toggle_timer_off.IN := FALSE;
	toggle_timer_on.IN  := FALSE;
	Q := FALSE;
END_IF;
END_FUNCTION_BLOCK

(* POU Standard FB's/FB_Motor_Ctrl, ST *)
(********************************************************************************************************

NAME...........	:	FB_Motor_Ctrl
DATE...........	:	5/20/2014
AUTHOR.........	:	SAMPLE

DESCRIPTION....	:	Function Block for Motor Drive

HISTORY:	
5/20/2014	v1.0.0	Start coding
*********************************************************************************************************)
FUNCTION_BLOCK FB_Motor_Ctrl
VAR_INPUT
	bRun					: BOOL; (* When high motor is commanded to turn on  *)
	bDrive_OK				: BOOL; (* True when drive has no faults			*)
	bDriveRunning			: BOOL; (* True when drive is running				*)
	nCommandedSpeed			: LREAL;(* Speed command from application			*)
END_VAR
VAR_OUTPUT
	bDrive_Enable			: BOOL; (* When true drive gets enable signal 	    *)
	nDriveSpeed				: LREAL;(* Speed Value for drive					*)

END_VAR

VAR
	SCALE_FACTOR			: REAL:= 2.0;
END_VAR
IF bDrive_OK THEN
	bDrive_Enable := bRun;
ELSE
	bDrive_Enable := FALSE;
END_IF;

(* If drive running then send speed *)
IF bDrive_Enable THEN
	nDriveSpeed := nCommandedSpeed * SCALE_FACTOR;
END_IF;

(* DEBUG REMOVE WHEN READY TODO:GPK*)
bDrive_Enable := bRun;
END_FUNCTION_BLOCK

(* POU Standard FB's/FB_CylinderControl, ST *)
FUNCTION_BLOCK FB_CylinderControl
VAR_INPUT
	bCylinder_Trigger	: BOOL;	(* Command to trigger cyliner 			*)
	bCylinder_Extended	: BOOL; (* True when cylinder fully extended 	*)
	bCylinder_Retracted : BOOL;	(* True when cylinder fully retracted	*)
	bEnable_Diagnostics : BOOL; (* When true diagnostics are enabled	*)
	tExtend_Timeout		: TIME; (* Time for extend timeout				*)
	tRetract_Timeout	: TIME; (* Time for retract tiemout				*)
	bReset				: BOOL; (* When true errors are reset			*)
	iConfiguration		: BYTE; (* Cylinder config. 0 = ext & ret sensors, 1 = Extend Sensor only, 2 = retract Sensor Only *)
END_VAR
VAR_OUTPUT
	bExtend_Cylinder	: BOOL;
	bRetract_Cylinder	: BOOL;
	bExtend_Error		: BOOL; (* True when an extend error is detected*)
	bRetract_Error		: BOOL; (* True when there is a retract error   *)
	bDevice_Home		: BOOL; (* True when device is home				*)
END_VAR
VAR
	RE_Trigger			: R_TRIG;
	RE_Extend_Sensor	: R_TRIG;
	RE_Retract_Sensor	: R_TRIG;

	TmrExtend			: TON;
	TmrRetract			: TON;
	TmrRetractOff		: TON;

END_VAR
(* Leading Edge Detection *)
RE_Trigger(CLK:= bCylinder_Trigger );
RE_Extend_Sensor(CLK:= bCylinder_Extended );
RE_Retract_Sensor(CLK:= bCylinder_Retracted );

(* Timers Serviced *)
TmrExtend(IN:= bExtend_Cylinder , PT:= tExtend_Timeout  );
TmrRetract(IN:= bRetract_Cylinder , PT:= tRetract_Timeout );
TmrRetractOff(PT:= tRetract_Timeout - T#500ms );

(* Check leading edge of trigger signal *)
IF RE_Trigger.Q THEN
	bExtend_Cylinder := TRUE;
	bRetract_Cylinder := FALSE;
END_IF;

CASE iConfiguration OF
	0: (* Extend and Retract Sensors *)
		(* Check leading edge of extend sensor *)
		IF RE_Extend_Sensor.Q THEN
			bExtend_Cylinder := FALSE;
			bRetract_Cylinder := TRUE;
		END_IF;

		(* Check leading edge of retract sensor *)
		IF RE_Retract_Sensor.Q THEN
			bExtend_Cylinder := FALSE;
			bRetract_Cylinder := FALSE;
		END_IF;
		(* Check if homed or not *)
		IF bCylinder_Retracted THEN
			bDevice_Home := TRUE;
		ELSE
			bDevice_Home := FALSE;
		END_IF;
	1: (* Extend only sensor *)
		(* Check leading edge of extend sensor *)
		IF RE_Extend_Sensor.Q THEN
			bExtend_Cylinder := FALSE;
			bRetract_Cylinder := TRUE;
		END_IF;

		IF TmrRetractOff.Q THEN
			bExtend_Cylinder := FALSE;
			bRetract_Cylinder := FALSE;
		END_IF;

    2: (* Retract only Sensor *)

		IF RE_Retract_Sensor.Q THEN
			bExtend_Cylinder := FALSE;
			bRetract_Cylinder := FALSE;
		END_IF;
		(* Check if homed or not *)
		IF bCylinder_Retracted THEN
			bDevice_Home := TRUE;
		ELSE
			bDevice_Home := FALSE;
		END_IF;
END_CASE;

(* Check timers *)

IF TmrExtend.Q AND bEnable_Diagnostics THEN
	bExtend_Error := TRUE;
	bExtend_Cylinder := FALSE;
END_IF;

IF TmrRetract.Q AND bEnable_Diagnostics THEN
	bRetract_Error := TRUE;
	bRetract_Cylinder := FALSE;
END_IF;

(* Reset Error Flags *)
IF bReset THEN
	bRetract_Error := FALSE;
	bExtend_error  := FALSE;
END_IF;
END_FUNCTION_BLOCK

(* POU Motion/FB_CoupleAxis, LD *)
FUNCTION_BLOCK FB_CoupleAxis
VAR_INPUT
	bCoupleAxis				: BOOL;
	bDeCoupleAxis			: BOOL;
END_VAR
VAR_OUTPUT
	bCoupled				: BOOL;     (* True when coupled			*)
END_VAR
VAR_IN_OUT
	Master : AXIS_REF;					(* axis reference data structure *)
	Slave : AXIS_REF;					(* axis reference data structure *)

END_VAR
VAR
	MC_GearIn				: MC_GearIn;				(* MC FB To gear in two axis						*)
	GearInOut				: ST_McOutputs;

	MC_GearOut				: MC_GearOut;				(* MC FB To gear out two axis						*)
	GearOutOut				: ST_McOutputs;

END_VAR
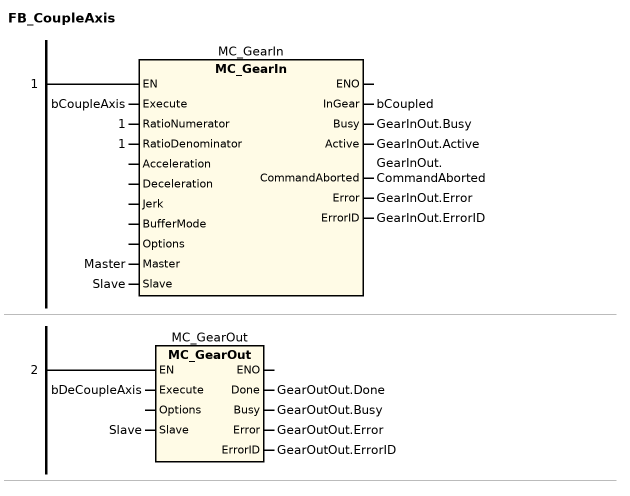
_LD_ (* Ladder Diagram *)
NETWORK 1
	*
		EN --- MC_GearIn:MC_GearIn(Execute: bCoupleAxis, RatioNumerator: 1, RatioDenominator: 1, Acceleration: , Deceleration: , Jerk: , BufferMode: , Options: , Master: Master, Slave: Slave, Busy => GearInOut.Busy, Active => GearInOut.Active, CommandAborted => GearInOut.CommandAborted, Error => GearInOut.Error, ErrorID => GearInOut.ErrorID) => bCoupled
NETWORK 2
	*
		EN --- MC_GearOut:MC_GearOut(Execute: bDeCoupleAxis, Options: , Slave: Slave, Busy => GearOutOut.Busy, Error => GearOutOut.Error, ErrorID => GearOutOut.ErrorID) => GearOutOut.Done
_END_LD_
END_FUNCTION_BLOCK

(* POU HMI, ST *)
PROGRAM HMI
VAR
	bHMIIncRecipe				: BOOL; (* Tied to HMI Button in receipe editor to increment current recipe *)
	bHMIDecRecipe				: BOOL; (* decrement current recipe											*)

	RE_bHMIIncRecipe    		: R_TRIG;(* Rising edge for increment recipe button							*)
	RE_bHMIDecRecipe			: R_TRIG;(* Rising edge for decrement recipe button							*)
	RE_bHMIIncMovePosition		: ARRAY[1..NUMBER_OF_AXIS] OF R_TRIG;(* Rising edge for button to move forward in recipe table for manual move*)
	RE_bHMIDecMovePosition		: ARRAY[1..NUMBER_OF_AXIS] OF R_TRIG;(* Rising edge for button to move bckward in recipe table for manual move*)

	bFaultReset					: BOOL; (* Fault reset 																	 *)

	bShowPopup					: BOOL; (* When true pop up is shown 													 *)
	bAtHomeScreen				: BOOL; (* True when at the home screen 												 *)
	bProgramError				: BOOL; (* True when there is a program selection Error									 *)

	bCutTimerError				: BOOL; (* True when the cutter timer in recipe is not set								 *)
	bNumberOfCutsRecipeError	: BOOL; (* True when the number fo cuts is not set correctly in recipe					 *)
	bMoveTable1Error			: ARRAY[1..NUMBER_OF_MOVES] OF BOOL; (* Each index is true when a move is zero			 *)
	bMoveTable2Error			: ARRAY[1..2] OF BOOL; (* Each index is true when a move is zero			 			 *)
	bMoveTable3Error			: ARRAY[1..2] OF BOOL; (* Each index is true when a move is zero			 			 *)
	bMoveTable4Error			: ARRAY[1..NUMBER_OF_MOVES] OF BOOL; (* Each index is true when a move is zero			 *)
	bMoveTable5Error			: ARRAY[1..2] OF BOOL; (* Each index is true when a move is zero			 			 *)
	bPartTypeNameRecipeError	: BOOL; (* True when no name given to a part type										 *)
	bSpeedSettingErrorAxis1		: BOOL; (* True when no speed set in recipe editor										 *)
	bSpeedSettingErrorAxis2		: BOOL; (* True when no speed set in recipe editor										 *)
	bSpeedSettingErrorAxis3		: BOOL; (* True when no speed set in recipe editor										 *)
	bSpeedSettingErrorAxis4		: BOOL; (* True when no speed set in recipe editor										 *)
	bSpeedSettingErrorAxis5		: BOOL; (* True when no speed set in recipe editor										 *)

	bHMIIncMovePosition			: ARRAY[1..NUMBER_OF_AXIS] OF BOOL; (* Increment flag for manual move screen 			 *)
	bHMIDecMovePosition			: ARRAY[1..NUMBER_OF_AXIS] OF BOOL; (* Decremet flag for the manual move screen 		 *)

	bHMIManMotionTablePos		: ARRAY[1..NUMBER_OF_AXIS] OF BYTE; (* Holds place in move table a manual motion move is *)
	loop						: BYTE; (* Used for the for loops *)

	nLeftSpindleXOffset			: LREAL; (* Used to drive the position of the axis on the mimic screen 					 *)
	nRightSpindleXOffset		: LREAL; (* Used to drive the position of the axis on the mimic screen 					 *)
	nCutterYOffset				: LREAL; (* Used to drive the position of the axis on the mimic screen 				 	 *)
	nCutterSlideXOffset			: LREAL; (* Used to drive the position of the axis on the mimic screen 				 	 *)
	nEnagageXOffset			    : LREAL; (* Used to drive the position of the axis on the mimic screen 					 *)

	AutoLogout					: FB_AutoLogout; (* Auto Logout User Function											 *)
END_VAR
RE_bHMIDecRecipe(CLK:= bHMIDecRecipe );
RE_bHMIIncRecipe(CLK:= bHMIINCRecipe );

(* Call auto logout routine, use this if you want the HMI to auto logout a user.*)
(* Set the level at which to start the timer, the delay time and which level to log into after timer has elapsed*)
AutoLogout(
	bEnabled:= TRUE ,
	timeLogoutTime:= T#10m,
	nLogoutLevel:= 4,
	nLogoutToLevel:= 1,
	CurrentUserLevel:= CurrentUserLevel);

(* Loop through number of axis to check rising edge of increment and decrement buttons *)
FOR loop := 1 TO NUMBER_OF_AXIS DO
	RE_bHMIIncMovePosition[loop](CLK:= bHMIIncMovePosition[loop] );
	RE_bHMIDecMovePosition[loop](CLK:= bHMIDecMovePosition[loop] );
END_FOR;

(* Check Recipe Number is Valid *)
IF nRecipeNumber < 1 OR nRecipeNumber > NUMBER_OF_RECIPES THEN
	nRecipeNumber := 1;
END_IF;

IF RE_bHMIDecRecipe.Q AND nRecipeNumber > 1 THEN
	nRecipeNumber := nRecipeNumber - 1;
END_IF;

IF RE_bHMIIncRecipe.Q AND nRecipeNumber < NUMBER_OF_RECIPES THEN
	nRecipeNumber := nRecipeNumber + 1;
END_IF;

(* Set at home screen flag if the current screen is the home screen *)
bAtHomeScreen := CurrentVisu = 'TC_VISU';


(* Manual Motion Screen Handler Axis 1 *)
IF RE_bHMIIncMovePosition[1].Q THEN
	IF bHMIManMotionTablePos[1] < (MachineRecipes[nCurrentRecipe].nNumberOfCuts + 1) THEN
		bHMIManMotionTablePos[1] := bHMIManMotionTablePos[1] + 1;
	END_IF;
	MAIN.nTargetPosition[1] := MachineRecipes[nCurrentRecipe].arrAxis1MoveTable[bHMIManMotionTablePos[1]];
	MAIN.nMoveVelocity[1] := 500;
END_IF;

IF RE_bHMIDecMovePosition[1].Q THEN
	IF bHMIManMotionTablePos[1] > 1 THEN
		bHMIManMotionTablePos[1] := bHMIManMotionTablePos[1] - 1;
	END_IF;
	MAIN.nTargetPosition[1] := MachineRecipes[nCurrentRecipe].arrAxis1MoveTable[bHMIManMotionTablePos[1]];
	MAIN.nMoveVelocity[1] := 500;
END_IF;


(* Manual Motion Screen Handler Axis 2 *)
IF RE_bHMIIncMovePosition[2].Q THEN
	IF bHMIManMotionTablePos[2] < 2 THEN
		bHMIManMotionTablePos[2] := bHMIManMotionTablePos[2] + 1;
	END_IF;
	MAIN.nTargetPosition[2] := MachineRecipes[nCurrentRecipe].arrAxis2MoveTable[bHMIManMotionTablePos[2]];
	MAIN.nMoveVelocity[2] := 500;
END_IF;

IF RE_bHMIDecMovePosition[2].Q THEN
	IF bHMIManMotionTablePos[2] > 1 THEN
		bHMIManMotionTablePos[2] := bHMIManMotionTablePos[2] - 1;
	END_IF;
	MAIN.nTargetPosition[2] := MachineRecipes[nCurrentRecipe].arrAxis2MoveTable[bHMIManMotionTablePos[2]];
	MAIN.nMoveVelocity[2] := 500;
END_IF;

(* Manual Motion Screen Handler Axis 3 *)
IF RE_bHMIIncMovePosition[3].Q THEN
	IF bHMIManMotionTablePos[3] < 2 THEN
		bHMIManMotionTablePos[3] := bHMIManMotionTablePos[3] + 1;
	END_IF;
	MAIN.nTargetPosition[3] := MachineRecipes[nCurrentRecipe].arrAxis3MoveTable[bHMIManMotionTablePos[3]];
	MAIN.nMoveVelocity[3] := 500;
END_IF;

IF RE_bHMIDecMovePosition[3].Q THEN
	IF bHMIManMotionTablePos[3] > 1 THEN
		bHMIManMotionTablePos[3] := bHMIManMotionTablePos[3] - 1;
	END_IF;
	MAIN.nTargetPosition[3] := MachineRecipes[nCurrentRecipe].arrAxis3MoveTable[bHMIManMotionTablePos[3]];
	MAIN.nMoveVelocity[3] := 500;
END_IF;


(* Manual Motion Screen Handler Axis 4 *)
IF RE_bHMIIncMovePosition[4].Q THEN
	IF bHMIManMotionTablePos[4] < (MachineRecipes[nCurrentRecipe].nNumberOfCuts + 1) THEN
		bHMIManMotionTablePos[4] := bHMIManMotionTablePos[4] + 1;
	END_IF;
	MAIN.nTargetPosition[4] := MachineRecipes[nCurrentRecipe].arrAxis4MoveTable[bHMIManMotionTablePos[4]];
	MAIN.nMoveVelocity[4] := 500;
END_IF;

IF RE_bHMIDecMovePosition[4].Q THEN
	IF bHMIManMotionTablePos[4] > 1 THEN
		bHMIManMotionTablePos[4] := bHMIManMotionTablePos[4] - 1;
	END_IF;
	MAIN.nTargetPosition[4] := MachineRecipes[nCurrentRecipe].arrAxis4MoveTable[bHMIManMotionTablePos[4]];
	MAIN.nMoveVelocity[4] := 500;
END_IF;

(* Manual Motion Screen Handler Axis 5 *)
IF RE_bHMIIncMovePosition[5].Q THEN
	IF bHMIManMotionTablePos[5] < 2 THEN
		bHMIManMotionTablePos[5] := bHMIManMotionTablePos[5] + 1;
	END_IF;
	MAIN.nTargetPosition[5] := MachineRecipes[nCurrentRecipe].arrAxis5MoveTable[bHMIManMotionTablePos[5]];
	MAIN.nMoveVelocity[5] := 500;
END_IF;

IF RE_bHMIDecMovePosition[5].Q THEN
	IF bHMIManMotionTablePos[5] > 1 THEN
		bHMIManMotionTablePos[5] := bHMIManMotionTablePos[5] - 1;
	END_IF;
	MAIN.nTargetPosition[5] := MachineRecipes[nCurrentRecipe].arrAxis5MoveTable[bHMIManMotionTablePos[5]];
	MAIN.nMoveVelocity[5] := 500;
END_IF;

	(* Assign Scaled values for the MIMIC Screens absolute move positions *)

	nLeftSpindleXOffset			:= MAIN.Axis[1].nActualPosition/10;
	nRightSpindleXOffset		:= MAIN.Axis[2].nActualPosition/10;
	nCutterYOffset				:= MAIN.Axis[3].nActualPosition/2;
	nCutterSlideXOffset			:= MAIN.Axis[4].nActualPosition/10;
	nEnagageXOffset			    := MAIN.Axis[5].nActualPosition/2;


(* Check we have a valid program *)
CASE nMachineType OF
	CUTTER:
		IF MachineRecipes[nCurrentRecipe].nNumberOfCuts > 0 AND MachineRecipes[nCurrentRecipe].arrAxis1MoveTable[1] > 0 AND MachineRecipes[nCurrentRecipe].arrAxis2MoveTable[1] > 0
		AND MachineRecipes[nCurrentRecipe].arrAxis3MoveTable[1] > 0 AND MachineRecipes[nCurrentRecipe].arrAxis4MoveTable[1] > 0 AND MachineRecipes[nCurrentRecipe].arrAxis5MoveTable[1] > 0 THEN
			bProgramError := FALSE;
		ELSE
			bProgramError := TRUE;
			faults.bProgramError := TRUE; (* Flag an Error to display a fault on the HMI *)
		END_IF;
	SIZER:
		IF MachineRecipes[nCurrentRecipe].nNumberOfCycles > 0 AND MachineRecipes[nCurrentRecipe].arrAxis1MoveTable[1] > 0 THEN
			bProgramError := FALSE;
		ELSE
			bProgramError := TRUE;
		END_IF;
END_CASE;



(* Receipe Checks Here *)
(* Code to validate bounds of receipe values *)
IF MachineRecipes[nRecipeNumber].timeCutterTimer < T#50ms THEN
	bCutTimerError := TRUE;
ELSE
	bCutTimerError := FALSE;
END_IF;

IF  MachineRecipes[nRecipeNumber].nNumberOfCuts > 0 THEN
	bNumberOfCutsRecipeError := FALSE;
ELSE
	bNumberOfCutsRecipeError := TRUE;
END_IF;

(* Loop throuch Axis 1 move table make sure it has valid data *)
FOR loop := 1 TO NUMBER_OF_MOVES DO
	IF MachineRecipes[nRecipeNumber].arrAxis1MoveTable[loop] = 0 THEN
		bMoveTable1Error[loop] := TRUE;
	ELSE
		bMoveTable1Error[loop] := FALSE;
	END_IF;
	IF MachineRecipes[nRecipeNumber].arrAxis4MoveTable[loop] = 0 THEN
		bMoveTable4Error[loop] := TRUE;
	ELSE
		bMoveTable4Error[loop] := FALSE;
	END_IF;
END_FOR;

FOR loop := 1 TO 2 DO
	IF MachineRecipes[nRecipeNumber].arrAxis2MoveTable[loop] = 0 THEN
		bMoveTable2Error[loop] := TRUE;
	ELSE
		bMoveTable2Error[loop] := FALSE;
	END_IF;
	IF MachineRecipes[nRecipeNumber].arrAxis3MoveTable[loop] = 0 THEN
		bMoveTable3Error[loop] := TRUE;
	ELSE
		bMoveTable3Error[loop] := FALSE;
	END_IF;
	IF MachineRecipes[nRecipeNumber].arrAxis5MoveTable[loop] = 0 THEN
		bMoveTable5Error[loop] := TRUE;
	ELSE
		bMoveTable5Error[loop] := FALSE;
	END_IF;
END_FOR;

(* Check Speed Setting *)
IF MachineRecipes[nRecipeNumber].rAxis1Speed = 0 THEN
	bSpeedSettingErrorAxis1 := TRUE;
ELSE
	bSpeedSettingErrorAxis1 := FALSE;
END_IF;

IF MachineRecipes[nRecipeNumber].rAxis2Speed = 0 THEN
	bSpeedSettingErrorAxis2 := TRUE;
ELSE
	bSpeedSettingErrorAxis2 := FALSE;
END_IF;

IF MachineRecipes[nRecipeNumber].rAxis3Speed = 0 THEN
	bSpeedSettingErrorAxis3 := TRUE;
ELSE
	bSpeedSettingErrorAxis3 := FALSE;
END_IF;

IF MachineRecipes[nRecipeNumber].rAxis4Speed = 0 THEN
	bSpeedSettingErrorAxis4 := TRUE;
ELSE
	bSpeedSettingErrorAxis4 := FALSE;
END_IF;

IF MachineRecipes[nRecipeNumber].rAxis5Speed = 0 THEN
	bSpeedSettingErrorAxis5 := TRUE;
ELSE
	bSpeedSettingErrorAxis5 := FALSE;
END_IF;

(* Check Recipe Name *)
IF MachineRecipes[nRecipeNumber].sRecipeName = '' THEN
	bPartTypeNameRecipeError := TRUE;
ELSE
	bPartTypeNameRecipeError := FALSE;
END_IF;
END_PROGRAM

(* POU Standard FB's/FB_AutoLogout, ST *)
(********************************************************************************************************
NAME...........	:	Auto Logout Function Block.
DATE...........	:	08.6.2010
AUTHOR.........	:	Graeme Peek 

DESCRIPTION....	:	Handles timer to auto log out user
HISTORY:	
08.11.2014	v1.1.0	GPK	Start coding
*********************************************************************************************************)
FUNCTION_BLOCK FB_AutoLogout
VAR_INPUT
	bEnabled					: BOOL;
	timeLogoutTime				: TIME;
	nLogoutLevel				: INT; (* The level which starts the timer 											*)
	nLogoutToLevel				: INT; (* The level at which to logout to  											*)
END_VAR
VAR_OUTPUT
END_VAR
VAR
	tmrLogoutTimer				: TON;  (* Timer to logout user after a set period 									*)
END_VAR
VAR_IN_OUT
	CurrentUserLevel 			: INT;
END_VAR
(* Logout timer called here *)
tmrLogoutTimer(IN:= (CurrentUserLevel > (nLogoutLevel - 1) AND bEnabled) , PT:= timeLogoutTime);

(* Once timer has elapse set the new user level *)
IF tmrLogoutTimer.Q THEN
	CurrentUserLevel := nLogoutToLevel;
END_IF;
END_FUNCTION_BLOCK

(* POU Machine, ST *)
PROGRAM Machine
VAR
	ErrorHandler				: FB_ErrorHandler;
	WarningHandler				: FB_WarningHandler;



END_VAR
ErrorHandler(
	guards_ok:= , 
	safety_enabled:= , 
	start_button:= , 
	reset_all_errors:= , 
	Faults:= Faults,
	bError_Present=> , 
	iError_Count=> , 
	bError_Detected=> , 
	arrActive_Errors=> ,
	sFirstError=> );

WarningHandler(
	reset_all_warnings:= , 
	Warnings:= Warnings,
	warning_present=> ,
	warning_count=> );



(* Reset automatic mode if there is a fault *)
IF ErrorHandler.bError_Present THEN
	bAutomaticMode := FALSE;
END_IF;

MAIN.bFaultPresent := ErrorHandler.bError_Present;


(* If first program is empty load receipe with defaults *)
IF  MachineRecipes[1].nNumberOfCycles = 0 AND MachineRecipes[1].arrAxis1MoveTable[1] = 0 THEN
	Machine.init();
END_IF;
END_PROGRAM
ACTION init:
(* Load Program 1 Defaults *)
(* Axis 1 First *)
MachineRecipes[1].arrAxis1MoveTable[1] := 500;
MachineRecipes[1].arrAxis1MoveTable[2] := 1000;
MachineRecipes[1].arrAxis1MoveTable[3] := 1500;
MachineRecipes[1].arrAxis1MoveTable[4] := 2000;
MachineRecipes[1].arrAxis1MoveTable[5] := 2500;
MachineRecipes[1].arrAxis1MoveTable[6] := 3000;
MachineRecipes[1].arrAxis1MoveTable[7] := 3500;
MachineRecipes[1].rAxis1Speed		   := 550;
(* Axis #2 *)
MachineRecipes[1].arrAxis2MoveTable[1] := 20;
MachineRecipes[1].arrAxis2MoveTable[2] := -3500;
MachineRecipes[1].rAxis2Speed		   := 550;
(* Axis #3 *)
MachineRecipes[1].arrAxis3MoveTable[1] := 20;
MachineRecipes[1].arrAxis3MoveTable[2] := 50;
MachineRecipes[1].rAxis3Speed		   := 550;
(* Axis #4 *)
MachineRecipes[1].arrAxis4MoveTable[1] := 500;
MachineRecipes[1].arrAxis4MoveTable[2] := 1000;
MachineRecipes[1].arrAxis4MoveTable[3] := 1500;
MachineRecipes[1].arrAxis4MoveTable[4] := 2000;
MachineRecipes[1].arrAxis4MoveTable[5] := 2500;
MachineRecipes[1].arrAxis4MoveTable[6] := 3000;
MachineRecipes[1].arrAxis4MoveTable[7] := 3500;
MachineRecipes[1].rAxis4Speed		   := 550;
(* Axis #5 *)
MachineRecipes[1].arrAxis5MoveTable[1] := 20;
MachineRecipes[1].arrAxis5MoveTable[2] := 100;
MachineRecipes[1].rAxis5Speed		   := 550;

MachineRecipes[1].nNumberOfCuts		   := 5;
MachineRecipes[1].sRecipeName		   := 'Part Type #1';
MachineRecipes[1].timeCutterTimer      := T#100ms;
END_ACTION

(* POU ERRPROC/FB_ErrorHandler, ST *)
(********************************************************************************************************
NAME...........	:	Error Handler Function Block 
DATE...........	:	08.6.2014
AUTHOR.........	:	Graeme Peek ()

DESCRIPTION....	:	Handling of errors for the Machine.

HISTORY:	
08.6.2014	v1.1.0	GPK	Start coding
*********************************************************************************************************)
FUNCTION_BLOCK FB_ErrorHandler
VAR
	error_test				: BOOL;
	loop					: BYTE;
	RE_Error_Detected		: R_TRIG;
	sError_Description		: STRING;
	arrError_List	    	: ARRAY[0..50] OF STRING;
END_VAR
VAR_OUTPUT
	bError_Present			: BOOL;
	iError_Count 			: BYTE;
	bError_Detected			: BOOL;
	arrActive_Errors	    : ARRAY[0..10] OF STRING;
	sFirstError				: STRING;
END_VAR
VAR_INPUT
	guards_ok				: BOOL;
	safety_enabled			: BOOL;
	start_button			: BOOL;
	reset_all_errors		: BOOL;
END_VAR
VAR_IN_OUT
	Faults					: FAULTS_STRUCT;
END_VAR
RE_Error_Detected(CLK:=bError_Present , Q=> bError_Detected );
(* Fill Error Text List *)
arrError_List[0] := 'Operator Stop';
arrError_List[1] := 'Left Hand Spindle VFD Fault';
arrError_List[2] := 'Right Hand Spindle VFD Fault';
arrError_List[3] := 'Program Fault';
arrError_List[4] := 'Left Hand Spindle Servo Fault';
arrError_List[5] := 'Right Hand Spindle Servo Fault';
arrError_List[6] := 'Cutter Servo Fault';
arrError_List[7] := 'Cutter Slide Servo Fault';
arrError_List[8] := 'Engage Servo Fault';
arrError_List[9] := 'Cycle Time Exceeded';


iError_count := 0; (* Reset the error count prior to checking error count *)
(* Loop throught the number of defined errors checking if each one is true or false *)
FOR loop := 0 TO (SIZEOF(Faults) - 1) DO
	MEMCPY(ADR(error_test),ADR(Faults) + loop,1);
	IF 	reset_all_errors OR (start_button AND safety_enabled AND guards_ok) THEN
		MEMSET(ADR(faults) + loop,0,1);
	ELSIF error_test THEN
			iError_count := iError_count + 1;
        	arrActive_Errors[iError_Count] := arrError_List[loop];
	END_IF;
END_FOR;

IF iError_Count > 0 THEN
	bError_Present := TRUE;
	(* If error has not been acknowledged by stop button assign screen to display *)
ELSE
	bError_Present := FALSE;
END_IF;
reset_all_errors  := FALSE;

sFirstError := arrActive_Errors[1];

(* On rising edge of an error change to main screen *)
IF RE_Error_Detected.Q THEN
	CurrentVisu := 'TC_VISU'; (* Change Visualization to Home Screen *)
END_IF;
END_FUNCTION_BLOCK

(* POU ERRPROC/FB_WarningHandler, ST *)
(********************************************************************************************************
NAME...........	:	Warning Handler Function Block For Case Packer 2014
DATE...........	:	5.20.2014
AUTHOR.........	:	Nate Brown (Staalkat International BV, USA)

DESCRIPTION....	:	Handling of errors for the Packer.

HISTORY:	
05.20.2014	v1.1.0	GPK	Start coding
*********************************************************************************************************)
FUNCTION_BLOCK FB_WarningHandler
VAR
	warning_test			: BOOL;
	loop					: BYTE;
END_VAR
VAR_OUTPUT
	warning_present			: BOOL;
	warning_count 			: BYTE;
END_VAR
VAR_INPUT
	reset_all_warnings		: BOOL;
END_VAR
VAR_IN_OUT
	Warnings				: WARNINGS_STRUCT;

END_VAR
warning_count := 0; (* Reset the warning count prior to checking error count *)
(* Loop throught the number of defined warnings checking if each one is true or false *)
FOR loop := 0 TO (SIZEOF(warnings) - 1) DO
	MEMCPY(ADR(warning_test),ADR(warnings) + loop,1);
	IF 	reset_all_warnings THEN
		MEMSET(ADR(warnings) + loop,0,1);
	ELSIF warning_test THEN
		warning_count := warning_count + 1;
	END_IF;
END_FOR;

IF warning_count > 0 THEN
	warning_present := TRUE;
ELSE
	warning_present := FALSE;
END_IF;
reset_all_warnings  := FALSE;
END_FUNCTION_BLOCK

(* POU WritePersistent, LD *)
PROGRAM WritePersistent
VAR
	UPS_Shutdown				: FB_S_UPS; 			(* UPS FB							 *)
	bPowerFailDetected			: BOOL;					(* True when power supply is removed *)
	eUPSState					: E_S_UPS_State;		(* State of UPS FB					 *)
END_VAR
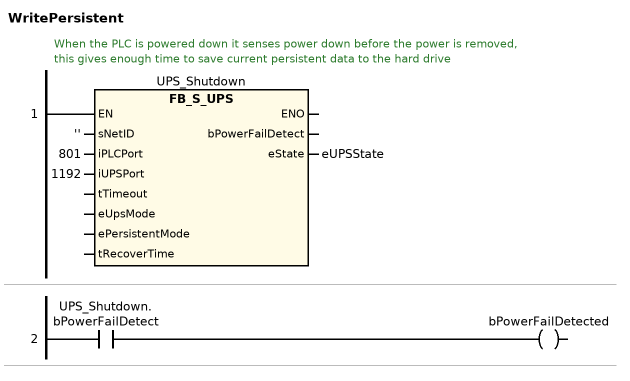
_LD_ (* Ladder Diagram *)
NETWORK 1 (* When the PLC is powered down it senses power down before the power is removed, / this gives enough time to save current persistent data to the hard drive *)
	*
		EN --- UPS_Shutdown:FB_S_UPS(sNetID: '', iPLCPort: 801, iUPSPort: 1192, tTimeout: , eUpsMode: , ePersistentMode: , tRecoverTime: , eState => eUPSState)
NETWORK 2
	[UPS_Shutdown.bPowerFailDetect] --- (bPowerFailDetected)
_END_LD_
(* the same logic as Structured Text *)
(* Network 1: see the listing above *)
(* Network 2 *)
bPowerFailDetected := UPS_Shutdown.bPowerFailDetect;
END_PROGRAM

(* POU Sequencer, ST *)
PROGRAM Sequencer
VAR
	nMachineSequence			: MACHINE_SEQUENCE; (* Holds Machine Sequence *)

	(* Delare Timers *)
	tmrCutterIn					: TON;
	tmrDelayCouple				: TON;

	nCurrentCutNumber			: BYTE; (* Current Cut Number *)
	bCutMade					: BOOL;
	bMoveLefttHandCommanded		: BOOL; (* Flag to ensure move command only issued once in a sequence step *)
	bMoveRightHandCommanded		: BOOL; (* Flag to ensure move command only issued once in a sequence step *)
	bMoveCutterSlideCommaned	: BOOL; (* Flag to ensure move command only issued once in a sequence step *)

	sSequence_Text				: STRING;

	bHMI_Overide				: BOOL; (* Temp test flag *)
	bHMI_ReturnAll				: BOOL; (* When true moves sequence to return all *)
	nSizerPosition				: BYTE; (* Position for sizer to be in *)
	nNumOfSizerCyclesCompleted  : BYTE;


	RE_MoveComplete				: R_TRIG;
END_VAR
tmrCutterIn(PT:= MachineRecipes[nCurrentRecipe].timeCutterTimer ); (* Call Cutter Timer *)
tmrDelayCouple(PT:= T#100ms );

(* Rising Edge Detection Handlers *)
RE_MoveComplete(CLK:= MAIN.bMoveAbsolute[SIZER_AXIS] );

CASE nMachineSequence OF


	MACHINE_INIT:
		tmrCutterIn.IN 					:= FALSE;
		MAIN.bCoupleAxis   				:= FALSE;
		MAIN.bDeCoupleAxis 				:= TRUE;
		MAIN.bLeftHandSpindleRun 	    := FALSE;
		MAIN.bRightHandSpindleRun		:= FALSE;
		nMachineSequence := MACHINE_READY;
	MACHINE_RESET:;
	MACHINE_FAULTED:;
	MACHINE_READY:
		MAIN.bDeCoupleAxis := FALSE;
		nCurrentCutNumber := 0; (* Reset Cut Counter *)
		MAIN.bInCycle := FALSE; (* Reset flag that machine is in cycle *)
		IF bAutomaticMode AND MAIN.bMachineRunning THEN
			CASE nMachineType OF
				CUTTER:
					IF ibCycleStartPB OR bHMI_Overide AND MachineRecipes[nCurrentRecipe].nNumberOfCuts > 0 THEN
						(* Clamp Part *)
						MAIN.bClosePartClamp := TRUE;
						IF ibPartClampLocked OR bHMI_Overide THEN
							nMachineSequence := ENABLE_SERVOS;
						END_IF;
					END_IF;
				SIZER:
					IF ibCycleStartPB OR bHMI_Overide AND MachineRecipes[nCurrentRecipe].nNumberOfCycles > 0 THEN
						(* Clamp Part *)
						IF MachineRecipes[nCurrentRecipe].bPartClampEnable THEN
							MAIN.bClosePartClamp := TRUE;
						END_IF;
						IF ibPartClampLocked OR bHMI_Overide THEN
							nMachineSequence := ENABLE_SERVOS;
						END_IF;
					END_IF;
			END_CASE;
		END_IF;
		MAIN.bInCycle := FALSE;
	ENABLE_SERVOS:
		CASE nMachineType OF
			CUTTER:
				(* Reset All Move Commands *)
				MAIN.bMoveAbsolute[LEFT_HAND_SPINDLE]	 := FALSE;
				MAIN.bMoveAbsolute[RIGHT_HAND_SPINDLE]	 := FALSE;
				MAIN.bMoveAbsolute[CUTTER_AXIS]	 		 := FALSE;
				MAIN.bMoveAbsolute[CUTTER_SLIDE]		 := FALSE;
				MAIN.bMoveAbsolute[ENGAGE_AXIS]	 		 := FALSE;
				(* Enable All Servos *)
				MAIN.bAxisEnable[LEFT_HAND_SPINDLE]  	 := TRUE;
				MAIN.bAxisEnable[RIGHT_HAND_SPINDLE] 	 := TRUE;
				MAIN.bAxisEnable[CUTTER_AXIS] 			 := TRUE;
				MAIN.bAxisEnable[CUTTER_SLIDE] 			 := TRUE;
				MAIN.bAxisEnable[ENGAGE_AXIS] 			 := TRUE;

				IF MAIN.Axis[1].bPowerOnStatus AND
				   MAIN.Axis[2].bPowerOnStatus AND
				   MAIN.Axis[3].bPowerOnStatus AND
				   MAIN.Axis[4].bPowerOnStatus AND
				   MAIN.Axis[5].bPowerOnStatus THEN
					nMachineSequence := MOVE_TO_END_CUT;
					bMoveRightHandCommanded := FALSE;
				END_IF;
			SIZER:
				(* Reset All Move Commands *)
				MAIN.bMoveAbsolute[SIZER_AXIS]	 := FALSE;
				MAIN.bMoveAbsolute[ARBOR_AXIS]	 := FALSE;
				MAIN.bAxisEnable[SIZER_AXIS] := TRUE;
				MAIN.bAxisEnable[ARBOR_AXIS] := TRUE;
				nNumOfSizerCyclesCompleted := 0;
				IF MAIN.Axis[SIZER_AXIS].bPowerOnStatus AND
				   	MAIN.Axis[ARBOR_AXIS].bPowerOnStatus THEN
						nMachineSequence := POSITION_SIZER_SERVOS;
				END_IF;
			END_CASE;

		POSITION_SIZER_SERVOS:

				(* Send Sizer to position *)
				MAIN.nTargetPosition[SIZER_AXIS]  := MachineRecipes[nCurrentRecipe].arrAxis1MoveTable[2];
				(* Make sure velocity is non zero use default if it is *)
				IF MachineRecipes[nCurrentRecipe].rAxis1Speed > 0 THEN
					MAIN.nMoveVelocity[SIZER_AXIS]	 := MachineRecipes[nCurrentRecipe].rAxis1Speed;
				ELSE
					MAIN.nMoveVelocity[SIZER_AXIS]	 := DEAFULT_AXIS_SPEED;
				END_IF;
				MAIN.bMoveAbsolute[SIZER_AXIS]	 := TRUE;

				(* Send Arbor Axis to Returned *)
				MAIN.nTargetPosition[ARBOR_AXIS]  := MachineRecipes[nCurrentRecipe].arrAxis2MoveTable[2];
				(* Make sure velocity is non zero use default if it is *)
				IF MachineRecipes[nCurrentRecipe].rAxis2Speed > 0 THEN
					MAIN.nMoveVelocity[ARBOR_AXIS]	 := MachineRecipes[nCurrentRecipe].rAxis1Speed;
				ELSE
					MAIN.nMoveVelocity[ARBOR_AXIS]	 := DEAFULT_AXIS_SPEED;
				END_IF;
				MAIN.bMoveAbsolute[ARBOR_AXIS]	 := TRUE;

				IF MAIN.Axis[SIZER_AXIS].bMoveComplete AND MAIN.Axis[ARBOR_AXIS].bMoveComplete THEN
					nMachineSequence := MOVE_TO_START_SIZER;
					MAIN.bMoveAbsolute[SIZER_AXIS]	 := FALSE;
					MAIN.bMoveAbsolute[ARBOR_AXIS]	 := FALSE;
					nSizerPosition := 3;
				END_IF;

	MOVE_TO_START_SIZER:

				(* Send Sizer to position *)
				MAIN.nTargetPosition[SIZER_AXIS]  := MachineRecipes[nCurrentRecipe].arrAxis1MoveTable[nSizerPosition];
				(* Make sure velocity is non zero use default if it is *)
				IF MachineRecipes[nCurrentRecipe].rAxis1Speed > 0 THEN
					MAIN.nMoveVelocity[SIZER_AXIS]	 := MachineRecipes[nCurrentRecipe].rAxis1Speed;
				ELSE
					MAIN.nMoveVelocity[SIZER_AXIS]	 := DEAFULT_AXIS_SPEED;
				END_IF;

				MAIN.bMoveAbsolute[SIZER_AXIS]	 := TRUE;
				IF MAIN.Axis[SIZER_AXIS].bMoveComplete THEN
					nMachineSequence := MOVE_TO_CRUSHED_POSITION;
					MAIN.bMoveAbsolute[SIZER_AXIS]	 := FALSE;
					nSizerPosition := nSizerPosition + 1;
				END_IF;


	MOVE_TO_CRUSHED_POSITION:
				(* Send Sizer to position *)
				MAIN.nTargetPosition[SIZER_AXIS]  := MachineRecipes[nCurrentRecipe].arrAxis1MoveTable[nSizerPosition];
				(* Make sure velocity is non zero use default if it is *)
				IF MachineRecipes[nCurrentRecipe].rAxis1Speed > 0 THEN
					MAIN.nMoveVelocity[SIZER_AXIS]	 := MachineRecipes[nCurrentRecipe].rAxis1Speed;
				ELSE
					MAIN.nMoveVelocity[SIZER_AXIS]	 := DEAFULT_AXIS_SPEED;
				END_IF;

				MAIN.bMoveAbsolute[SIZER_AXIS]	 := TRUE;
				IF MAIN.Axis[SIZER_AXIS].bMoveComplete THEN
					nMachineSequence := MOVE_SIZER_TO_RELIEVED_POSITION;
					MAIN.bMoveAbsolute[SIZER_AXIS]	 := FALSE;
					nSizerPosition := nSizerPosition + 1;
				END_IF;

	MOVE_SIZER_TO_RELIEVED_POSITION:

				(* Send Sizer to position *)
				MAIN.nTargetPosition[SIZER_AXIS]  := MachineRecipes[nCurrentRecipe].arrAxis1MoveTable[nSizerPosition];
				(* Make sure velocity is non zero use default if it is *)
				IF MachineRecipes[nCurrentRecipe].rAxis1Speed > 0 THEN
					MAIN.nMoveVelocity[SIZER_AXIS]	 := MachineRecipes[nCurrentRecipe].rAxis1Speed;
				ELSE
					MAIN.nMoveVelocity[SIZER_AXIS]	 := DEAFULT_AXIS_SPEED;
				END_IF;

				MAIN.bMoveAbsolute[SIZER_AXIS]	 := TRUE;

				IF MAIN.Axis[SIZER_AXIS].bMoveComplete THEN
					IF nNumOfSizerCyclesCompleted < MachineRecipes[nCurrentRecipe].nNumberOfCycles THEN
						nMachineSequence := MOVE_TO_CRUSHED_POSITION;
						nSizerPosition := nSizerPosition - 1;
						MAIN.bMoveAbsolute[SIZER_AXIS]	 := FALSE;
					ELSE
						nMachineSequence := MOVE_SIZER_TO_UNLOAD;
						MAIN.bMoveAbsolute[SIZER_AXIS]	 := FALSE;
					END_IF;
				END_IF;
				IF RE_MoveComplete.Q THEN
					nNumOfSizerCyclesCompleted := nNumOfSizerCyclesCompleted + 1;
				END_IF;
	MOVE_SIZER_TO_UNLOAD:

				(* Send Sizer to position *)
				MAIN.nTargetPosition[SIZER_AXIS]  := MachineRecipes[nCurrentRecipe].arrAxis1MoveTable[1];
				(* Make sure velocity is non zero use default if it is *)
				IF MachineRecipes[nCurrentRecipe].rAxis1Speed > 0 THEN
					MAIN.nMoveVelocity[SIZER_AXIS]	 := MachineRecipes[nCurrentRecipe].rAxis1Speed;
				ELSE
					MAIN.nMoveVelocity[SIZER_AXIS]	 := DEAFULT_AXIS_SPEED;
				END_IF;

				MAIN.bMoveAbsolute[SIZER_AXIS]	 := TRUE;

				IF MAIN.Axis[SIZER_AXIS].bMoveComplete THEN
						MAIN.bMoveAbsolute[SIZER_AXIS]	 := FALSE;
					MAIN.bClosePartClamp := FALSE;
					IF MAIN.Axis_REF[SIZER_AXIS].NcToPlc.ActPos = MachineRecipes[nCurrentRecipe].arrAxis1MoveTable[4] THEN
						nMachineSequence := RETURN_SIZER;
					END_IF;
				END_IF;

	RETURN_SIZER:
				(* Send Sizer to return position *)
				MAIN.nTargetPosition[SIZER_AXIS]  := MachineRecipes[nCurrentRecipe].arrAxis1MoveTable[1];
				(* Make sure velocity is non zero use default if it is *)
				IF MachineRecipes[nCurrentRecipe].rAxis1Speed > 0 THEN
					MAIN.nMoveVelocity[SIZER_AXIS]	 := MachineRecipes[nCurrentRecipe].rAxis1Speed;
				ELSE
					MAIN.nMoveVelocity[SIZER_AXIS]	 := DEAFULT_AXIS_SPEED;
				END_IF;

				MAIN.nTargetPosition[ARBOR_AXIS]  := MachineRecipes[nCurrentRecipe].arrAxis2MoveTable[1];
				(* Make sure velocity is non zero use default if it is *)
				IF MachineRecipes[nCurrentRecipe].rAxis2Speed > 0 THEN
					MAIN.nMoveVelocity[ARBOR_AXIS]	 := MachineRecipes[nCurrentRecipe].rAxis2Speed;
				ELSE
					MAIN.nMoveVelocity[ARBOR_AXIS]	 := DEAFULT_AXIS_SPEED;
				END_IF;

				MAIN.bMoveAbsolute[SIZER_AXIS]	 := TRUE;
				MAIN.bMoveAbsolute[ARBOR_AXIS]	 := TRUE;

				IF MAIN.Axis[SIZER_AXIS].bMoveComplete AND MAIN.Axis[ARBOR_AXIS].bMoveComplete THEN
					MAIN.bMoveAbsolute[SIZER_AXIS]	 := FALSE;
					MAIN.bMoveAbsolute[ARBOR_AXIS]	 := FALSE;
					nMachineSequence := MACHINE_READY;
				END_IF;


	MOVE_TO_END_CUT:
		MAIN.bInCycle := TRUE;
		nCurrentCutNumber := 1; (* Reset Cut Counter *)
		(* Left Hand Spindle Servo Advances to end cut position *)
		MAIN.nTargetPosition[LEFT_HAND_SPINDLE]  := MachineRecipes[nCurrentRecipe].arrAxis1MoveTable[2];
		IF MachineRecipes[nCurrentRecipe].rAxis1Speed > 0 THEN
			MAIN.nMoveVelocity[LEFT_HAND_SPINDLE]	 := MachineRecipes[nCurrentRecipe].rAxis1Speed;
		ELSE
			MachineRecipes[nCurrentRecipe].rAxis1Speed := DEAFULT_AXIS_SPEED;
			MAIN.nMoveVelocity[LEFT_HAND_SPINDLE]	 := DEAFULT_AXIS_SPEED;
		END_IF;
		IF MAIN.Axis[RIGHT_HAND_SPINDLE].bMoveComplete THEN
			MAIN.bMoveAbsolute[LEFT_HAND_SPINDLE]	 := TRUE;
			MAIN.bMoveAbsolute[RIGHT_HAND_SPINDLE]	 := FALSE;
		END_IF;
		(* Move Right hand spindle out of the way *)
		MAIN.nTargetPosition[RIGHT_HAND_SPINDLE]  := MachineRecipes[nCurrentRecipe].arrAxis2MoveTable[1];
		IF  MachineRecipes[nCurrentRecipe].rAxis2Speed > 0 THEN
			MAIN.nMoveVelocity[RIGHT_HAND_SPINDLE]	 := MachineRecipes[nCurrentRecipe].rAxis2Speed;
		ELSE
			MachineRecipes[nCurrentRecipe].rAxis2Speed := DEAFULT_AXIS_SPEED;
			MAIN.nMoveVelocity[RIGHT_HAND_SPINDLE]	 := DEAFULT_AXIS_SPEED;
		END_IF;
		IF (NOT bMoveRightHandCommanded) THEN
			MAIN.bMoveAbsolute[RIGHT_HAND_SPINDLE]	 := TRUE;
		END_IF;
		(*Move Cutter Slide to first position *)
		MAIN.nTargetPosition[CUTTER_SLIDE]  := MachineRecipes[nCurrentRecipe].arrAxis4MoveTable[2];
		IF MachineRecipes[nCurrentRecipe].rAxis4Speed > 0 THEN
			MAIN.nMoveVelocity[CUTTER_SLIDE]	:= MachineRecipes[nCurrentRecipe].rAxis4Speed;
		ELSE
			MachineRecipes[nCurrentRecipe].rAxis4Speed := DEAFULT_AXIS_SPEED;
			MAIN.nMoveVelocity[CUTTER_SLIDE]	:= DEAFULT_AXIS_SPEED;
		END_IF;
		MAIN.bMoveAbsolute[CUTTER_SLIDE]	:= TRUE;

		(* Once left spindle and right spindle have completed move to advance engage axis *)
		IF MAIN.Axis[LEFT_HAND_SPINDLE].bMoveComplete AND MAIN.Axis[RIGHT_HAND_SPINDLE].bMoveComplete THEN
			MAIN.bMoveAbsolute[LEFT_HAND_SPINDLE] := FALSE;
			bMoveRightHandCommanded := FALSE;
			MAIN.bMoveAbsolute[CUTTER_SLIDE]	:= FALSE;
			nMachineSequence     	:= ADVANCE_ENGAGE;
		END_IF;

		(* Reset move command once move is completed *)
		IF MAIN.Axis[CUTTER_AXIS].bMoveComplete THEN
			MAIN.bMoveAbsolute[CUTTER_AXIS] := FALSE;
		END_IF;

	COUPLE_DRIVES:
		MAIN.bDeCoupleAxis := FALSE;
		IF MAIN.Axis_REF[2].NcToPlc.ActVelo = 0 THEN
			tmrDelayCouple.IN := TRUE;
		ELSE
			tmrDelayCouple.IN := FALSE;
		END_IF;
		IF MAIN.Axis_REF[2].NcToPlc.ActVelo = 0 AND MAIN.Axis_REF[4].NcToPlc.ActVelo = 0 AND tmrDelayCouple.Q AND bAutomaticMode THEN
			MAIN.bCoupleAxis := TRUE;
		END_IF;

		IF MAIN.bAxis2Coupled AND bAutomaticMode (*AND MAIN.bAxis4Coupled*) THEN
			nMachineSequence := MOVE_TO_NEXT_CUT;
			bMoveLefttHandCommanded := FALSE; (* Ensure move command flags are reset *)
			bMoveRightHandCommanded := FALSE;
			tmrDelayCouple.IN 		:= FALSE;
		END_IF;

	DECOUPLE_DRIVES:
		MAIN.bCoupleAxis   := FALSE;
		MAIN.bDeCoupleAxis := TRUE;
		MAIN.bMoveAbsolute[CUTTER_AXIS] := FALSE;
		nMachineSequence   := RETURN_MACHINE;
		nPartsCounter := nPartsCounter + 1;

	MOVE_TO_NEXT_CUT:

		MAIN.nTargetPosition[LEFT_HAND_SPINDLE]  := MachineRecipes[nCurrentRecipe].arrAxis1MoveTable[nCurrentCutNumber + 1] ;
		MAIN.nMoveVelocity[LEFT_HAND_SPINDLE]	 := MachineRecipes[nCurrentRecipe].rAxis1Speed;
		IF (NOT bMoveLefttHandCommanded) AND MAIN.bMachineRunning THEN
			MAIN.bMoveAbsolute[LEFT_HAND_SPINDLE]	 := TRUE;
			bMoveLefttHandCommanded					 := TRUE;
		END_IF;

		(* If Drives not coupled Then*)
		IF NOT MAIN.bAxis2Coupled (*AND NOT MAIN.bAxis4Coupled*) AND MAIN.bMachineRunning THEN
			MAIN.nTargetPosition[RIGHT_HAND_SPINDLE] := MachineRecipes[nCurrentRecipe].arrAxis2MoveTable[nCurrentCutNumber] ;
			MAIN.nMoveVelocity[RIGHT_HAND_SPINDLE]	 := MachineRecipes[nCurrentRecipe].rAxis2Speed;
			IF MAIN.Axis[LEFT_HAND_SPINDLE].bMoveComplete AND (NOT bMoveRightHandCommanded) THEN
				MAIN.bMoveAbsolute[RIGHT_HAND_SPINDLE]	 := TRUE;
				bMoveRightHandCommanded					 := TRUE;
			END_IF;

			(* If this second cut then couple drives*)
			IF nCurrentCutNumber = 2 AND ( bMoveLefttHandCommanded AND (NOT MAIN.Axis_REF[1].Status.HasJob)) AND ( bMoveRightHandCommanded
				AND (NOT MAIN.Axis_REF[2].Status.HasJob)) AND bAutomaticMode AND MAIN.bMachineRunning THEN
				(* COUPLE DRIVES *);
				nMachineSequence := COUPLE_DRIVES;
				bMoveLefttHandCommanded := FALSE;
				bMoveRightHandCommanded := FALSE;
			END_IF;
		END_IF;

		(*Move Cutter Slide to next position *)
		MAIN.nTargetPosition[CUTTER_SLIDE]  := MachineRecipes[nCurrentRecipe].arrAxis4MoveTable[nCurrentCutNumber + 1];
		IF MachineRecipes[nCurrentRecipe].rAxis4Speed > 0 THEN
			MAIN.nMoveVelocity[CUTTER_SLIDE]	:= MachineRecipes[nCurrentRecipe].rAxis4Speed;
		ELSE
			MachineRecipes[nCurrentRecipe].rAxis4Speed := DEAFULT_AXIS_SPEED;
			MAIN.nMoveVelocity[CUTTER_SLIDE]	:= DEAFULT_AXIS_SPEED;
		END_IF;

		IF (NOT bMoveCutterSlideCommaned) THEN
			MAIN.bMoveAbsolute[CUTTER_SLIDE]	:= TRUE;
			bMoveCutterSlideCommaned 			:= TRUE;
		END_IF;

		IF MAIN.bAxis2Coupled (*AND MAIN.bAxis4Coupled*) THEN
			IF MAIN.Axis[LEFT_HAND_SPINDLE].bMoveComplete (*AND MAIN.Axis[CUTTER_SLIDE].bMoveComplete*) THEN
				bMoveLefttHandCommanded  := FALSE;
				bMoveRightHandCommanded  := FALSE;
				bMoveCutterSlideCommaned := FALSE;
				nMachineSequence     	 := ADVANCE_ENGAGE;
			END_IF;
		END_IF;

	ADVANCE_ENGAGE:

		MAIN.bMoveAbsolute[ENGAGE_AXIS]	 	  := TRUE;
		(* Advance the Engage *)
		MAIN.nTargetPosition[ENGAGE_AXIS]  := MachineRecipes[nCurrentRecipe].arrAxis5MoveTable[2];
		IF MachineRecipes[nCurrentRecipe].rAxis5Speed > 0 THEN
			MAIN.nMoveVelocity[ENGAGE_AXIS]	 := MachineRecipes[nCurrentRecipe].rAxis5Speed;
		ELSE
			MachineRecipes[nCurrentRecipe].rAxis5Speed := DEAFULT_AXIS_SPEED;
			MAIN.nMoveVelocity[ENGAGE_AXIS]	 := DEAFULT_AXIS_SPEED;
		END_IF;

		IF MAIN.Axis[ENGAGE_AXIS].bMoveComplete THEN
			MAIN.bMoveAbsolute[ENGAGE_AXIS]	 := FALSE;
			nMachineSequence     			 := OPERATE_CUT;
			bCutMade			 			 := FALSE;
		END_IF;

	RETURN_ENGAGE:

		MAIN.bMoveAbsolute[ENGAGE_AXIS]	 	  := TRUE;
		(* Advance the Engage *)
		MAIN.nTargetPosition[ENGAGE_AXIS]  := MachineRecipes[nCurrentRecipe].arrAxis5MoveTable[1];
		IF MachineRecipes[nCurrentRecipe].rAxis5Speed > 0 THEN
			MAIN.nMoveVelocity[ENGAGE_AXIS]	 := MachineRecipes[nCurrentRecipe].rAxis5Speed;
		ELSE
			MachineRecipes[nCurrentRecipe].rAxis5Speed := DEAFULT_AXIS_SPEED;
			MAIN.nMoveVelocity[ENGAGE_AXIS]	 := DEAFULT_AXIS_SPEED;
		END_IF;

		IF MAIN.Axis[ENGAGE_AXIS].bMoveComplete THEN
			MAIN.bMoveAbsolute[ENGAGE_AXIS]	 := FALSE;
			nMachineSequence     			 := MOVE_TO_NEXT_CUT;
			bMoveLefttHandCommanded 		 := FALSE; (* Ensure move command flags are reset *)
			bMoveRightHandCommanded 		 := FALSE;
			bCutMade			 			 := FALSE;
		END_IF;


	OPERATE_CUT:
		MAIN.nTargetPosition[CUTTER_AXIS]  := MachineRecipes[nCurrentRecipe].arrAxis3MoveTable[2];
		IF MachineRecipes[nCurrentRecipe].rAxis3Speed > 0 THEN
			MAIN.nMoveVelocity[CUTTER_AXIS]	 := MachineRecipes[nCurrentRecipe].rAxis3Speed;
		ELSE
			MachineRecipes[nCurrentRecipe].rAxis3Speed := DEAFULT_AXIS_SPEED;
			MAIN.nMoveVelocity[CUTTER_AXIS]	 := MachineRecipes[nCurrentRecipe].rAxis3Speed;
		END_IF;
		IF (NOT bCutMade) THEN
			MAIN.bMoveAbsolute[CUTTER_AXIS]	 := TRUE;
			bCutMade := TRUE;
		END_IF;
		IF MAIN.Axis[CUTTER_AXIS].bMoveComplete AND (NOT MAIN.bMoveAbsolute[CUTTER_AXIS]) THEN
			MAIN.bMoveAbsolute[CUTTER_AXIS] := FALSE;
			(* Ensure we have some reasonable value for a time delay if not put default value in *)
			IF MachineRecipes[nCurrentRecipe].timeCutterTimer < T#50ms THEN
				MachineRecipes[nCurrentRecipe].timeCutterTimer := T#500ms;
			END_IF;
			tmrCutterIn.IN := TRUE; (* Start delay timer *)
		END_IF;
		(* Once Cutter timer has been reached move on *)
		IF tmrCutterIn.Q THEN
			tmrCutterIn.IN := FALSE;
			bCutMade := FALSE;
			nMachineSequence := RETRACT_FROM_CUT;
		END_IF;

		MAIN.bLeftHandSpindleRun 			  := TRUE; (* Turn on spindle VFD*)
		IF MAIN.bAxis2Coupled THEN
			MAIN.bRightHandSpindleRun		  := TRUE;
		END_IF;

	RETRACT_FROM_CUT:
		MAIN.nTargetPosition[CUTTER_AXIS]  := MachineRecipes[nCurrentRecipe].arrAxis3MoveTable[1] ;
		MAIN.nMoveVelocity[CUTTER_AXIS]	 := MachineRecipes[nCurrentRecipe].rAxis3Speed;
		MAIN.bMoveAbsolute[CUTTER_AXIS]	 := TRUE;
		IF MAIN.Axis[CUTTER_AXIS].bMoveComplete THEN
			MAIN.bLeftHandSpindleRun 	    := FALSE;
			MAIN.bMoveAbsolute[CUTTER_AXIS] := FALSE;
			MAIN.bRightHandSpindleRun		:= FALSE;
			IF nCurrentCutNumber = machineRecipes[nCurrentRecipe].nNumberOfCuts THEN
				nMachineSequence := DECOUPLE_DRIVES;
			ELSE
				nCurrentCutNumber := nCurrentCutNumber + 1;
				nMachineSequence := RETURN_ENGAGE;
			END_IF;
		END_IF;

	RETURN_MACHINE:

		MAIN.nTargetPosition[LEFT_HAND_SPINDLE]  := MachineRecipes[nCurrentRecipe].arrAxis1MoveTable[1];
		IF MachineRecipes[nCurrentRecipe].rAxis1Speed > 0 THEN
			MAIN.nMoveVelocity[LEFT_HAND_SPINDLE]	 := MachineRecipes[nCurrentRecipe].rAxis1Speed;
		ELSE
			MachineRecipes[nCurrentRecipe].rAxis1Speed := DEAFULT_AXIS_SPEED;
			MAIN.nMoveVelocity[LEFT_HAND_SPINDLE]	 := DEAFULT_AXIS_SPEED;
		END_IF;

		(* Move Right hand spindle out of the way *)
		MAIN.nTargetPosition[RIGHT_HAND_SPINDLE]  := MachineRecipes[nCurrentRecipe].arrAxis2MoveTable[1];
		IF  MachineRecipes[nCurrentRecipe].rAxis2Speed > 0 THEN
			MAIN.nMoveVelocity[RIGHT_HAND_SPINDLE]	 := MachineRecipes[nCurrentRecipe].rAxis2Speed;
		ELSE
			MachineRecipes[nCurrentRecipe].rAxis2Speed := DEAFULT_AXIS_SPEED;
			MAIN.nMoveVelocity[RIGHT_HAND_SPINDLE]	 := DEAFULT_AXIS_SPEED;
		END_IF;

		(* Make Sure Cutter is Returned *)
		MAIN.nTargetPosition[CUTTER_AXIS]  := MachineRecipes[nCurrentRecipe].arrAxis3MoveTable[1];
		(* Make sure velocity is non zero use default if it is *)
		IF MachineRecipes[nCurrentRecipe].rAxis3Speed > 0 THEN
			MAIN.nMoveVelocity[CUTTER_AXIS]	 := MachineRecipes[nCurrentRecipe].rAxis3Speed;
		ELSE
			MAIN.nMoveVelocity[CUTTER_AXIS]	 := DEAFULT_AXIS_SPEED;
		END_IF;

		(* Return Cutter Slide *)
		MAIN.nTargetPosition[CUTTER_SLIDE]  := MachineRecipes[nCurrentRecipe].arrAxis4MoveTable[1];
		IF MachineRecipes[nCurrentRecipe].rAxis4Speed > 0 THEN
			MAIN.nMoveVelocity[CUTTER_SLIDE]	:= MachineRecipes[nCurrentRecipe].rAxis4Speed;
		ELSE
			MachineRecipes[nCurrentRecipe].rAxis4Speed := DEAFULT_AXIS_SPEED;
			MAIN.nMoveVelocity[CUTTER_SLIDE]	:= DEAFULT_AXIS_SPEED;
		END_IF;

		(* Set Return Engage Axis Position *)
		MAIN.nTargetPosition[ENGAGE_AXIS]  := MachineRecipes[nCurrentRecipe].arrAxis5MoveTable[1];
		IF MachineRecipes[nCurrentRecipe].rAxis5Speed > 0 THEN
			MAIN.nMoveVelocity[ENGAGE_AXIS]	 := MachineRecipes[nCurrentRecipe].rAxis5Speed;
		ELSE
			MachineRecipes[nCurrentRecipe].rAxis5Speed := DEAFULT_AXIS_SPEED;
			MAIN.nMoveVelocity[ENGAGE_AXIS]	 := DEAFULT_AXIS_SPEED;
		END_IF;


		IF MAIN.Axis[LEFT_HAND_SPINDLE].bMoveComplete AND MAIN.Axis[RIGHT_HAND_SPINDLE].bMoveComplete AND MAIN.Axis[CUTTER_AXIS].bMoveComplete AND
		  MAIN.Axis[CUTTER_SLIDE].bMoveComplete AND MAIN.Axis[ENGAGE_AXIS].bMoveComplete THEN
			nMachineSequence := MACHINE_READY;
		END_IF;

		(* Turn on drives in sequence required *)

		MAIN.bMoveAbsolute[ENGAGE_AXIS]	 		 := TRUE;

		IF MAIN.Axis_REF[ENGAGE_AXIS].NcToPlc.ActPos = MachineRecipes[nCurrentRecipe].arrAxis5MoveTable[1] THEN
			MAIN.bMoveAbsolute[CUTTER_AXIS]	 		 := TRUE;
		END_IF;

		IF MAIN.Axis_REF[CUTTER_AXIS].NcToPlc.ActPos = MachineRecipes[nCurrentRecipe].arrAxis3MoveTable[1] THEN
			MAIN.bMoveAbsolute[LEFT_HAND_SPINDLE]	 := TRUE;
			MAIN.bMoveAbsolute[RIGHT_HAND_SPINDLE]	 := TRUE;
			MAIN.bMoveAbsolute[CUTTER_SLIDE]		 := TRUE;
		END_IF;
		MAIN.bLeftHandSpindleRun 				 := FALSE;


END_CASE;

sSequence_Text := GetMachineSequenceActionDescription(iSequence_state := nMachineSequence);

IF bHMI_ReturnAll THEN
	nMachineSequence := RETURN_MACHINE;
END_IF;
END_PROGRAM

(* POU GetMachineSequenceActionDescription, ST *)
(********************************************************************************************************
NAME...........	:	GetMotionSequenceActionDescription
DATE...........	:	06.04.2014
AUTHOR.........	:	Graeme Peek (Beckhoff Automation)

DESCRIPTION....	:	Function to assign meaningful text to action text based on current action

HISTORY:	
06.04.2014	v1.0.0	GPK	Start coding
*********************************************************************************************************)
FUNCTION GetMachineSequenceActionDescription : STRING
VAR_INPUT
	iSequence_State 			: MACHINE_SEQUENCE;
END_VAR
VAR
END_VAR
CASE iSequence_State OF

	MACHINE_INIT:				GetMachineSequenceActionDescription := 'Initializing';
	MACHINE_RESET:				GetMachineSequenceActionDescription := 'Machine Reset';
	MACHINE_FAULTED:			GetMachineSequenceActionDescription := 'Machine Faulted';
	MACHINE_READY:	    		GetMachineSequenceActionDescription := 'Machine Ready';
	ENABLE_SERVOS:	  	 		GetMachineSequenceActionDescription := 'Enabling Servos';
	MOVE_TO_END_CUT:	  		GetMachineSequenceActionDescription := 'Move to end Cut';
	MOVE_TO_START_SIZER: 		GetMachineSequenceActionDescription := 'Move To Start Sizer';
	POSITION_SIZER_SERVOS:		GetMachineSequenceActionDescription := 'Position Sizer Servos';
	MOVE_TO_FIRST_CUT:			GetMachineSequenceActionDescription := 'Move to first cut';
	MOVE_TO_CRUSHED_POSITION:   GetMachineSequenceActionDescription := 'Move To Crushed Sizer Position';
	MOVE_SIZER_TO_RELIEVED_POSITION:GetMachineSequenceActionDescription := 'Move To Relaxed Position';
	MOVE_SIZER_TO_UNLOAD:       GetMachineSequenceActionDescription := 'Move Sizer To Unload Position';
	RETURN_SIZER:               GetMachineSequenceActionDescription := 'Return Sizer';
	COUPLE_DRIVES:				GetMachineSequenceActionDescription := 'Couple Drives';
	DECOUPLE_DRIVES:			GetMachineSequenceActionDescription := 'DeCouple Drives';
	OPERATE_FIRST_CUT:			GetMachineSequenceActionDescription := 'Operate First Cut';
	MOVE_TO_NEXT_CUT:			GetMachineSequenceActionDescription := 'Move To Next Cut';
	ADVANCE_ENGAGE:				GetMachineSequenceActionDescription := 'Advance Engage';
	RETURN_ENGAGE:				GetMachineSequenceActionDescription := 'Return Enagage';
	OPERATE_CUT:				GetMachineSequenceActionDescription := 'Operate Cut';
	RETRACT_FROM_CUT:			GetMachineSequenceActionDescription := 'Retract From Cut';
	RETURN_MACHINE:				GetMachineSequenceActionDescription := 'Return Machine';
ELSE
	GetMachineSequenceActionDescription := 'Unknown Sequence State';
END_CASE
END_FUNCTION

(* Visualisation MOTION SCREENS/ALL_AXIS
embedded screen at (2,0)-(0,127): dynamic style 
29 elements of other kinds (tables, trends, ...) not read
*)

(* Visualisation Helpers/Motion Helpers/AXIS
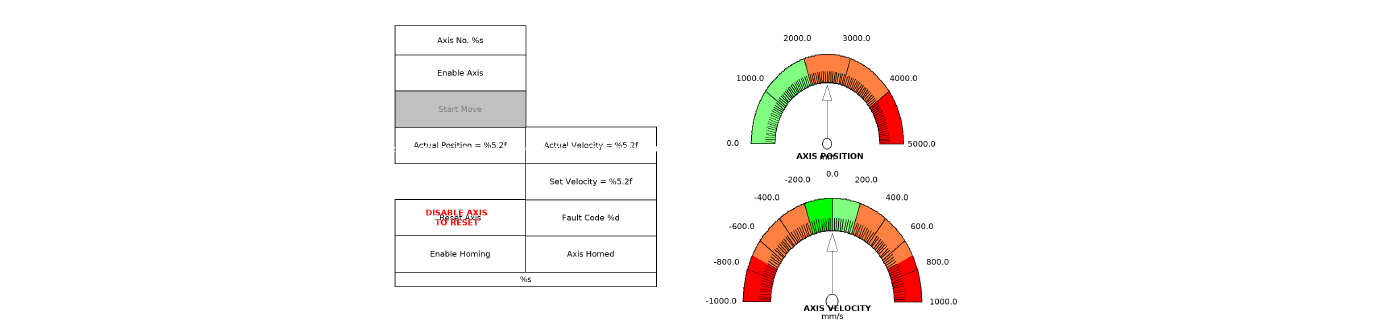
rectangle at (10,100)-(191,151): text "Start Move"; invisible if (NOT $InputDisable$); alarm colour if $MoveCommand$; toggles $MoveCommand$
rectangle at (10,150)-(191,201): text "Actual Position = %5.2f"; shows $AxisPosition$
rectangle at (10,50)-(191,101): text "Enable Axis"; alarm colour if $EnableAxis$; toggles $EnableAxis$
rectangle at (10,10)-(191,51): text "Axis No. %s"; shows $AxisNumber$; alarm colour if $AxisError$
rectangle at (10,100)-(191,151): text "Start Move"; invisible if $InputDisable$
rectangle at (10,250)-(191,301): text "Reset Axis"; invisible if $AxisError$ AND $EnableAxis$; taps $ResetAxis$
rectangle at (10,350)-(371,371): text "%s"; shows $AxisState$
rectangle at (10,300)-(191,351): text "Enable Homing"; alarm colour if $EnableHoming$; toggles $EnableHoming$
rectangle at (190,150)-(371,201): text "Actual Velocity = %5.2f"; shows $AxisVelocity$
rectangle at (190,300)-(371,351): text "Axis Homed"; alarm colour if $AxisHomed$
rectangle at (190,250)-(371,301): text "Fault Code %d"; shows $FaultCode$; alarm colour if $FaultCode$ > 0
group at (430,180)-(791,421)
  rectangle at (0,0)-(1,1): text "{ExtendedElement},Visu\ElementDLL.ete,0,@Zeigerinstrument,361,180,0,0,255,255,255,0,$VELOCITY$,mm/s,%.1f,0,1,1,20,200,-1000,1000,0,0,0,0,0,0,0,-13,80,400,Courier New,1,6,0,200,128,255,128,200,700,255,128,64,700,1000,255,0,0,-1000,-700,255,0,0,-700,-200,255,128,64,-200,0,0,255,0,0,255,255,255,,"
  rectangle at (2,172)-(58,188): text "-1000.0"
  rectangle at (13,126)-(61,142): text "-800.0"
  rectangle at (34,84)-(82,100): text "-600.0"
  rectangle at (68,50)-(116,66): text "-400.0"
  rectangle at (110,29)-(158,45): text "-200.0"
  rectangle at (169,22)-(193,38): text "0.0"
  rectangle at (207,29)-(247,45): text "200.0"
  rectangle at (249,50)-(289,66): text "400.0"
  rectangle at (283,84)-(323,100): text "600.0"
  rectangle at (304,126)-(344,142): text "800.0"
  rectangle at (308,173)-(356,189): text "1000.0"
  rectangle at (165,190)-(197,206): text "mm/s"
  polygon at (173,100)-(188,181): angle (($VELOCITY$ * 1.0)-0) * 0.09
rectangle at (450,380)-(791,421): text "AXIS VELOCITY"
rectangle at (190,200)-(371,251): text "Set Velocity = %5.2f"; shows $SetVelocity$
rectangle at (0,240)-(191,311): text "DISABLE AXIS / TO RESET"; invisible if NOT ($AxisError$ AND $EnableAxis$)
group at (450,-10)-(761,201)
  rectangle at (0,0)-(1,1): text "{ExtendedElement},Visu\ElementDLL.ete,0,@Zeigerinstrument,311,180,0,0,255,255,255,0,$AxisPosition$,mm,%.1f,0,1,1,50,1000,0,5000,0,0,0,0,0,0,0,-13,80,400,Courier New,1,3,0,2000,128,255,128,2000,4000,255,128,64,4000,5000,255,0,0,0,255,255,255,,"
  rectangle at (14,147)-(38,163): text "0.0"
  rectangle at (26,71)-(74,87): text "1000.0"
  rectangle at (91,24)-(139,40): text "2000.0"
  rectangle at (172,24)-(220,40): text "3000.0"
  rectangle at (237,71)-(285,87): text "4000.0"
  rectangle at (262,148)-(310,164): text "5000.0"
  rectangle at (148,163)-(164,179): text "mm"
  polygon at (149,87)-(162,156): angle (($AxisPosition$ * 1.0)-2500) * 0.036
rectangle at (440,170)-(781,211): text "AXIS POSITION"
embedded screen at (210,11)-(421,48): LED
embedded screen at (210,40)-(331,76): LED
embedded screen at (210,70)-(331,107): LED
embedded screen at (210,100)-(331,137): LED
218 more shapes without text or variables
1 elements of other kinds (tables, trends, ...) not read
*)

(* Visualisation MOTION SCREENS/AXIS1
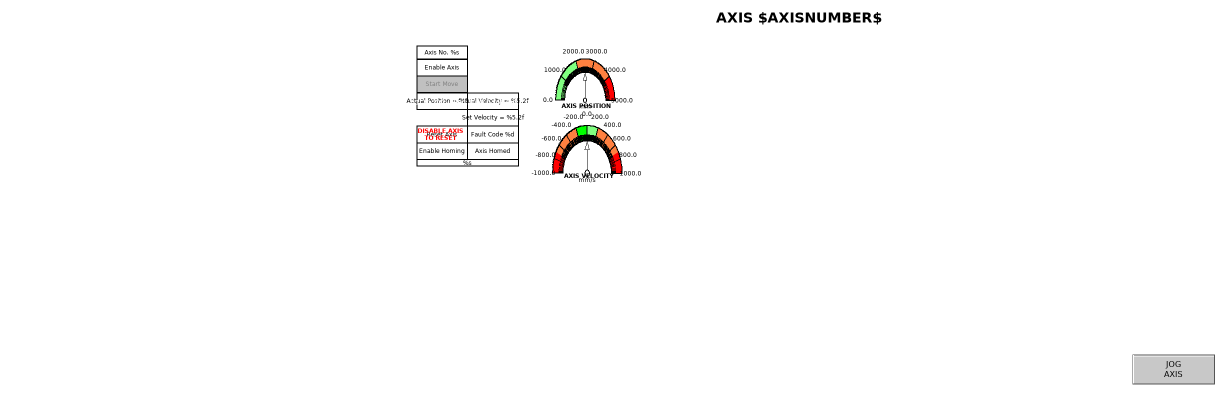
embedded screen at (0,0)-(801,381): AXIS_VISU
*)

(* Visualisation MOTION SCREENS/AXIS2
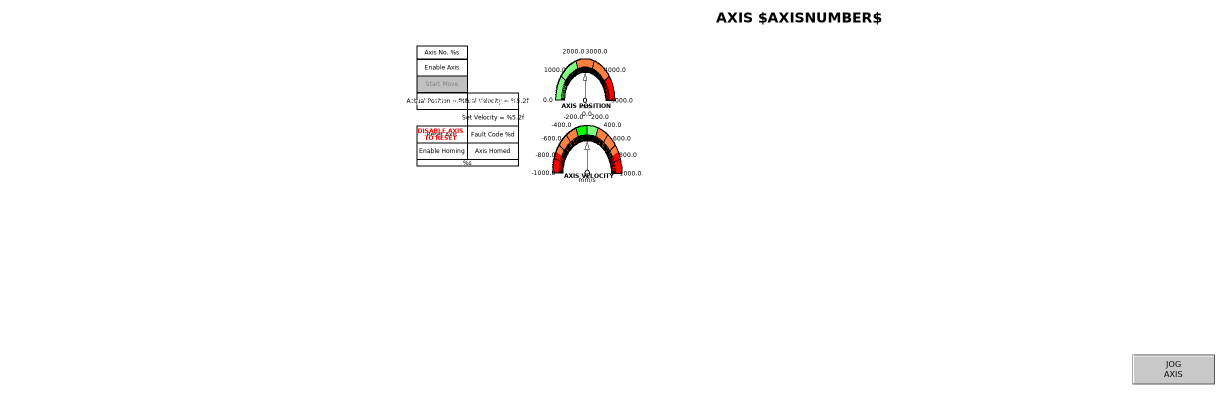
embedded screen at (0,0)-(801,381): AXIS_VISU
*)

(* Visualisation MOTION SCREENS/AXIS3
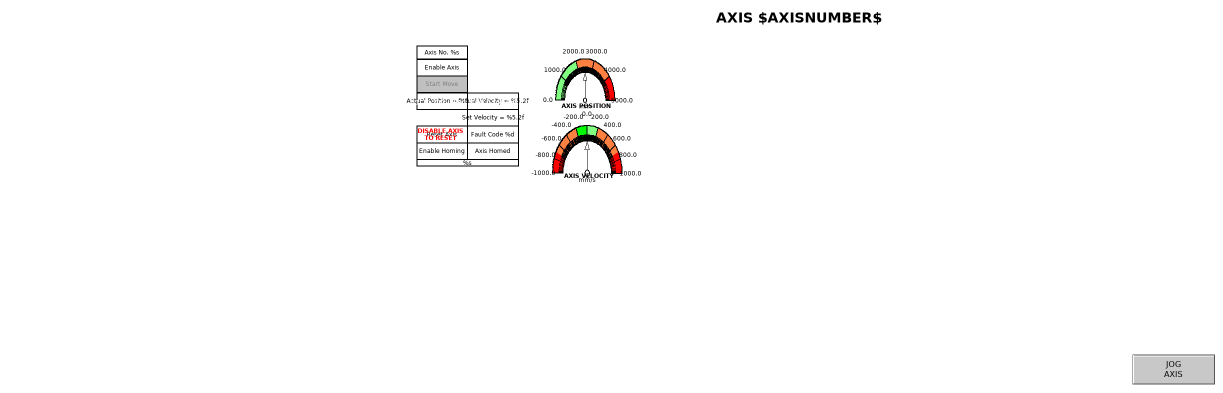
embedded screen at (0,0)-(801,381): AXIS_VISU
*)

(* Visualisation MOTION SCREENS/AXIS4
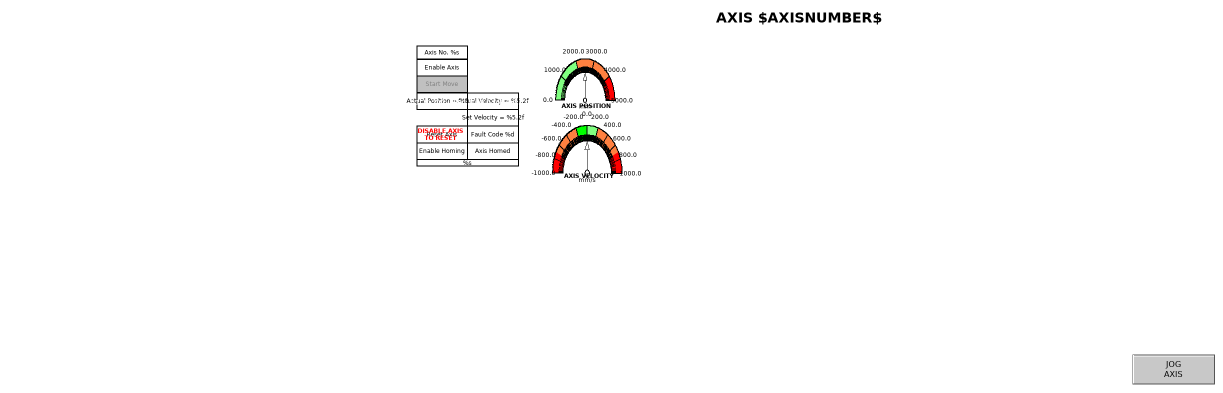
embedded screen at (0,0)-(801,381): AXIS_VISU
*)

(* Visualisation MOTION SCREENS/AXIS5
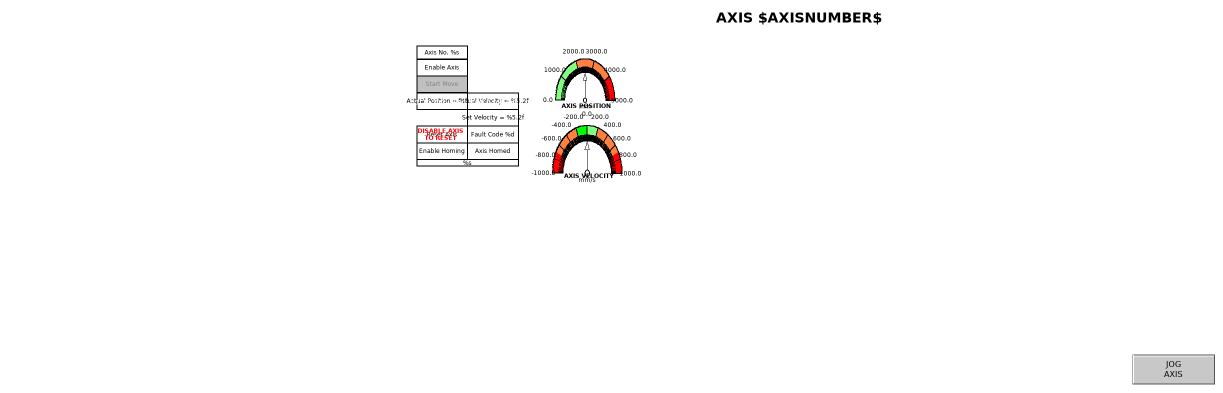
embedded screen at (0,0)-(801,381): AXIS_VISU
*)

(* Visualisation Helpers/Motion Helpers/AXIS_LITE
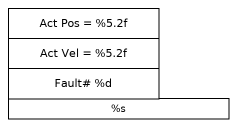
rectangle at (0,0)-(151,31): text "Act Pos = %5.2f"; shows $AxisPosition$; alarm colour if $EnableAxis$
rectangle at (0,90)-(221,111): text "%s"; shows $AxisState$
rectangle at (0,30)-(151,61): text "Act Vel = %5.2f"; shows $AxisVelocity$
rectangle at (0,60)-(151,91): text "Fault# %d"; shows $FaultCode$; invisible if $FaultCode$ = 0; alarm colour if $FaultCode$ > 0
*)

(* Visualisation Helpers/Motion Helpers/AXIS_VISU
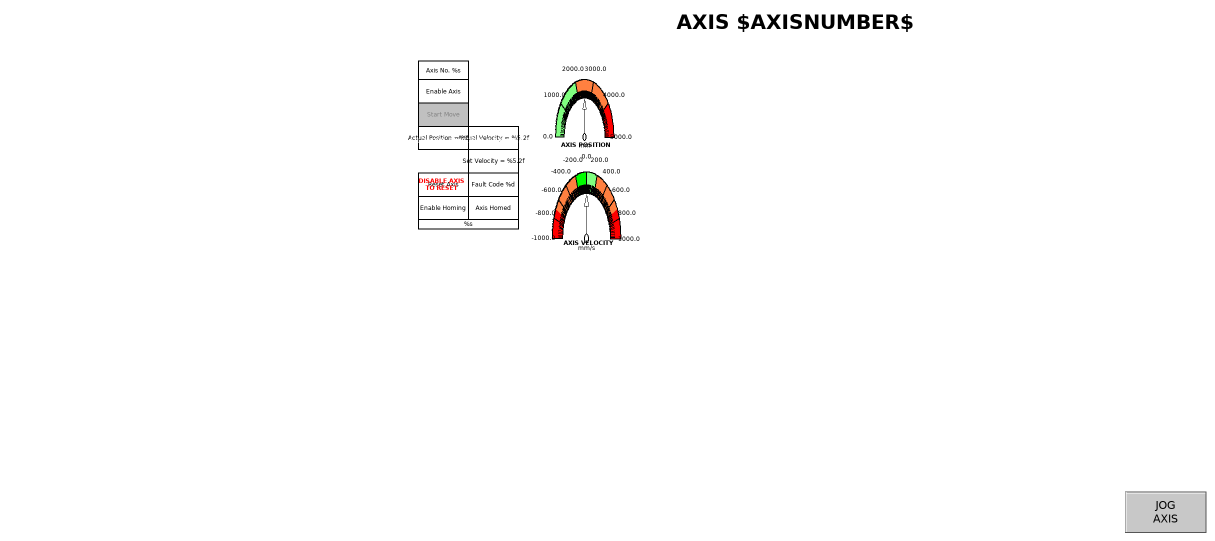
embedded screen at (0,50)-(221,251): Axis
rectangle at (210,0)-(551,41): text "AXIS $AXISNUMBER$"
button at (710,490)-(791,531): text "JOG / AXIS"; opens $JOG_AXIS$
*)

(* Visualisation Helpers/Buttons/Round_Buttons/GREEN_IND_BTN_BMP_MOMENTRY
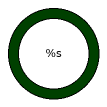
ellipse at (0,0)-(91,91): alarm colour if $INDICATOR$
ellipse at (10,10)-(81,81): text "%s"; shows $SWITCH_TITLE$; taps $SWITCH_INPUT$
*)

(* Visualisation Helpers/Buttons/Round_Buttons/GREEN_IND_BTN_BMP_TOGGLE
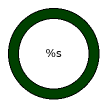
ellipse at (0,0)-(91,91): alarm colour if $INDICATOR$
ellipse at (10,10)-(81,81): text "%s"; shows $SWITCH_TITLE$; toggles $SWITCH_INPUT$
*)

(* Visualisation Helpers/Buttons/Round_Buttons/GRN_PUSH
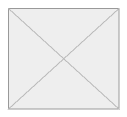
bitmap at (0,0)-(111,101): greenup.bmp
bitmap at (0,0)-(111,101): greendown.bmp
*)

(* Visualisation IO_SCREEN
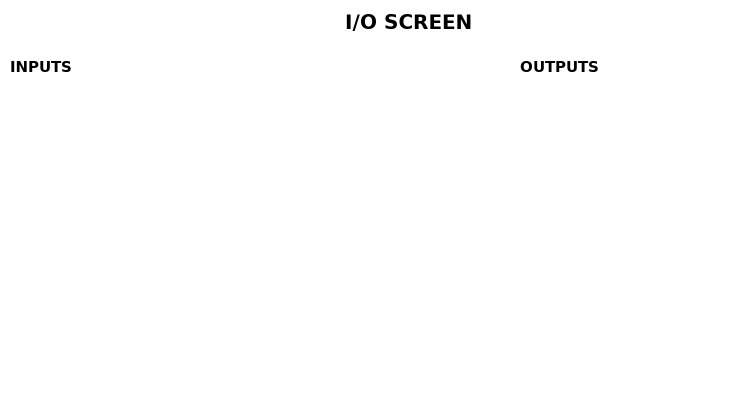
rounded rectangle at (20,90)-(231,121): text "Power On"; alarm colour if .ibPowerOn
rounded rectangle at (20,120)-(231,151): text "Light Screen Clear"; alarm colour if .ibLightScreenClear
rounded rectangle at (20,150)-(231,181): text "Cycle Start PB"; alarm colour if .ibCycleStartPB
rounded rectangle at (20,180)-(231,211): text "Left Hand Spindle Drive On"; alarm colour if .ibLeftHandSpindleDriveOn
rounded rectangle at (20,210)-(231,241): text "Left Hand Spindle Drive OK"; alarm colour if .ibLeftHandSpindleDriveOK
rounded rectangle at (20,240)-(231,271): text "Right Hand Spindle Drive On"; alarm colour if .ibRightHandSpindleDriveOn
rounded rectangle at (20,270)-(231,301): text "Right Hand Spindle Drive OK"; alarm colour if .ibRightHandSpindleDriveOK
rounded rectangle at (20,300)-(231,331): text "Part Clamp Advanced"; alarm colour if .ibPartClampAdvanced
rounded rectangle at (20,330)-(231,361): text "Part Clamp Returned"; alarm colour if .ibPartClampReturned
rounded rectangle at (20,360)-(231,391): text "Part Clamp Locked"; alarm colour if .ibPartClampLocked
rounded rectangle at (240,90)-(451,121): text "Hydraulics Overload"; alarm colour if .ibHydraulicsOverload
rectangle at (10,50)-(141,81): text "INPUTS"
rounded rectangle at (520,90)-(731,121): text "Left Hand Spindle Drive On"; alarm colour if .qbLeftHandSpindleOn
rounded rectangle at (520,120)-(731,151): text "Right Hand Spindle Drive On"; alarm colour if .qbRightHandSpindleOn
rounded rectangle at (520,150)-(731,181): text "Close Part Clamp Sol A"; alarm colour if .qbClosePartClampSolA
rounded rectangle at (520,180)-(731,211): text "Open Part Clamp Sol B"; alarm colour if .qbOpenPartClampSolB
rounded rectangle at (520,210)-(731,241): text "Spare"; alarm colour if .qbSpareOutput
rounded rectangle at (520,240)-(731,271): text "Green Lamp"; alarm colour if .qbOKToEnterGreenLamp
rounded rectangle at (520,270)-(731,301): text "Red Lamp"; alarm colour if .qbMachineInCycleFaultRedLamp
rectangle at (520,50)-(651,81): text "OUTPUTS"
rectangle at (320,0)-(501,41): text "I/O SCREEN"
11 more shapes without text or variables
*)

(* Visualisation Helpers/Motion Helpers/JOG_AXIS
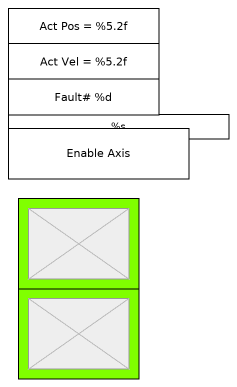
embedded screen at (10,320)-(131,411): RED_IND_SWITCH_BMP_MOMENTRY
embedded screen at (10,230)-(131,321): RED_IND_SWITCH_BMP_MTRY_LEFT
embedded screen at (0,40)-(221,171): AXIS_LITE
rectangle at (0,160)-(181,211): text "Enable Axis"; alarm colour if MAIN.bAxisEnable[$AXISNUMBER$]; toggles MAIN.bAxisEnable[$AXISNUMBER$]
*)

(* Visualisation MOTION SCREENS/JOG_AXIS1_3
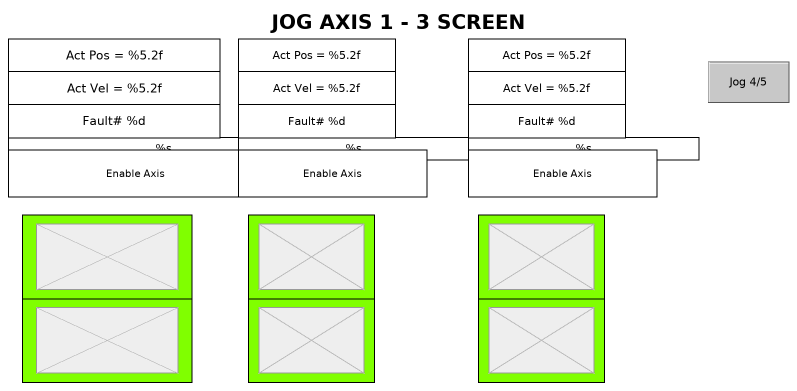
embedded screen at (0,0)-(311,381): JOG_AXIS
embedded screen at (230,0)-(461,381): JOG_AXIS
embedded screen at (460,0)-(691,381): JOG_AXIS
button at (700,60)-(781,101): text "Jog 4/5"; invisible if .nMachineType = SIZER; opens JOG_AXIS4_5
rectangle at (230,0)-(551,41): text "JOG AXIS 1 - 3 SCREEN"
*)

(* Visualisation MOTION SCREENS/JOG_AXIS4_5
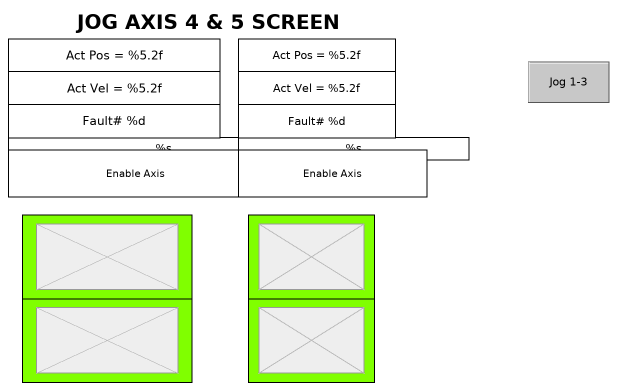
embedded screen at (180,0)-(491,381): JOG_AXIS
embedded screen at (410,0)-(641,381): JOG_AXIS
button at (700,60)-(781,101): text "Jog 1-3"; opens JOG_AXIS1_3
rectangle at (220,0)-(541,41): text "JOG AXIS 4 & 5 SCREEN"
*)

(* Visualisation Helpers/LED
ellipse at (0,5)-(21,26): alarm colour if $LED_STATE$
rectangle at (30,0)-(351,31): text "%s"; shows $LED_TITLE$
*)

(* Visualisation Helpers/Motion Helpers/MAN_AXIS
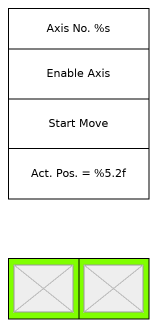
rectangle at (0,90)-(141,141): text "Start Move"; alarm colour if $MoveCommand$; toggles $MoveCommand$
rectangle at (0,140)-(141,191): text "Act. Pos. = %5.2f"; shows $AxisPosition$
rectangle at (0,40)-(141,91): text "Enable Axis"; alarm colour if $EnableAxis$; toggles $EnableAxis$
rectangle at (0,0)-(141,41): text "Axis No. %s"; shows $AxisNumber$
embedded screen at (70,250)-(141,311): RED_IND_SWITCH_BMP_MOMENTRY
embedded screen at (0,250)-(71,311): RED_IND_SWITCH_BMP_MTRY_LEFT
2 elements of other kinds (tables, trends, ...) not read
*)

(* Visualisation Helpers/Motion Helpers/MANUAL_MOTION
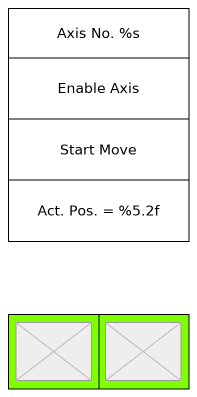
embedded screen at (0,-10)-(181,371): MAN_AXIS
*)

(* Visualisation MOTION SCREENS/MANUAL_MOTIONS
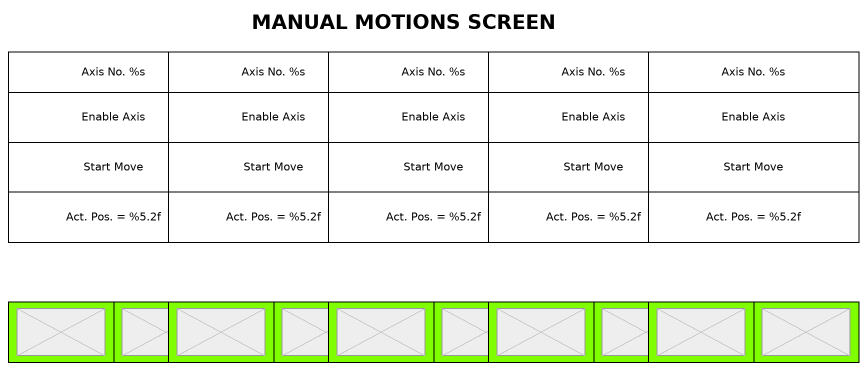
embedded screen at (0,50)-(211,361): MANUAL_MOTION
embedded screen at (160,50)-(371,361): MANUAL_MOTION
embedded screen at (320,50)-(531,361): MANUAL_MOTION
embedded screen at (480,50)-(691,361): MANUAL_MOTION
embedded screen at (640,50)-(851,361): MANUAL_MOTION
rectangle at (220,0)-(571,41): text "MANUAL MOTIONS SCREEN"
*)

(* Visualisation MIMIC
